LIN {X 0,Y 303.729,Z 621.055,A -85,B 0,C 180,E1 -15926.02,E2 -15926.02} C_VEL
LIN {X 0,Y 303.689,Z 622.489,A -85,B 0,C 180,E1 -15927.347,E2 -15927.347} C_VEL
LIN {X 0,Y 303.724,Z 623.5,A -85,B 0,C 180,E1 -15928.674,E2 -15928.674} C_VEL
LIN {X 0,Y 303.767,Z 624.114,A -85,B 0,C 180,E1 -15930,E2 -15930} C_VEL
LIN {X 0,Y 303.684,Z 624.33,A -85,B 0,C 180,E1 -15931.326,E2 -15931.326} C_VEL
LIN {X 0,Y 303.657,Z 624.123,A -85,B 0,C 180,E1 -15932.653,E2 -15932.653} C_VEL
LIN {X 0,Y 303.664,Z 623.508,A -85,B 0,C 180,E1 -15933.981,E2 -15933.981} C_VEL
LIN {X 0,Y 303.694,Z 622.179,A -85,B 0,C 180,E1 -15935.678,E2 -15935.678} C_VEL
LIN {X 0,Y 303.95,Z 619.276,A -85,B 0,C 180,E1 -15937.974,E2 -15937.974} C_VEL
LIN {X 0,Y 304.417,Z 615.707,A -85,B 0,C 180,E1 -15939.971,E2 -15939.971} C_VEL
LIN {X 0,Y 305.168,Z 611.059,A -85,B 0,C 180,E1 -15941.962,E2 -15941.962} C_VEL
LIN {X 0,Y 306.657,Z 604.076,A -85,B 0,C 180,E1 -15944.262,E2 -15944.262} C_VEL
LIN {X 0,Y 308.071,Z 596.828,A -85,B 0,C 180,E1 -15946.159,E2 -15946.159} C_VEL
LIN {X 0,Y 309.648,Z 588.913,A -85,B 0,C 180,E1 -15947.842,E2 -15947.842} C_VEL
LIN {X 0,Y 311.444,Z 579.671,A -85,B 0,C 180,E1 -15949.441,E2 -15949.441} C_VEL
LIN {X 0,Y 313.381,Z 569.416,A -85,B 0,C 180,E1 -15950.855,E2 -15950.855} C_VEL
LIN {X 0,Y 315.305,Z 558.079,A -85,B 0,C 180,E1 -15952.094,E2 -15952.094} C_VEL
LIN {X 0,Y 316.995,Z 546.32,A -85,B 0,C 180,E1 -15953.087,E2 -15953.087} C_VEL
LIN {X 0,Y 318.457,Z 533.399,A -85,B 0,C 180,E1 -15953.88,E2 -15953.88} C_VEL
LIN {X 0,Y 319.476,Z 519.67,A -85,B 0,C 180,E1 -15954.446,E2 -15954.446} C_VEL
LIN {X 0,Y 321.398,Z 456.74,A -85,B 0,C 180,E1 -15955.903,E2 -15955.903} C_VEL
LIN {X 0,Y 317.843,Z 434.507,A -85,B 0,C 180,E1 -15956.863,E2 -15956.863} C_VEL
LIN {X 0,Y 313.385,Z 414.246,A -85,B 0,C 180,E1 -15957.906,E2 -15957.906} C_VEL
LIN {X 0,Y 311.826,Z 410.324,A -85,B 0,C 180,E1 -15958.212,E2 -15958.212} C_VEL
LIN {X 0,Y 309.683,Z 400.252,A -85,B 0,C 180,E1 -15961.463,E2 -15961.463} C_VEL
LIN {X 0,Y 307.323,Z 390.367,A -85,B 0,C 180,E1 -15964.869,E2 -15964.869} C_VEL
LIN {X 0,Y 305.492,Z 383.429,A -85,B 0,C 180,E1 -15967.459,E2 -15967.459} C_VEL
LIN {X 0,Y 305.477,Z 383.421,A -85,B 0,C 180,E1 -15971.85,E2 -15971.85} C_VEL
LIN {X 0,Y 305.47,Z 383.432,A -85,B 0,C 180,E1 -15975.496,E2 -15975.496} C_VEL
LIN {X 0,Y 305.491,Z 383.43,A -85,B 0,C 180,E1 -15978.152,E2 -15978.152} C_VEL
LIN {X 0,Y 305.515,Z 383.43,A -85,B 0,C 180,E1 -15981.604,E2 -15981.604} C_VEL
LIN {X 0,Y 305.458,Z 383.435,A -85,B 0,C 180,E1 -15984.886,E2 -15984.886} C_VEL
LIN {X 0,Y 305.447,Z 383.436,A -85,B 0,C 180,E1 -15988.354,E2 -15988.354} C_VEL
LIN {X 0,Y 305.523,Z 383.423,A -85,B 0,C 180,E1 -15991.114,E2 -15991.114} C_VEL
LIN {X 0,Y 305.565,Z 383.413,A -85,B 0,C 180,E1 -15994.088,E2 -15994.088} C_VEL
LIN {X 0,Y 305.494,Z 383.421,A -85,B 0,C 180,E1 -15998.403,E2 -15998.403} C_VEL
LIN {X 0,Y 305.584,Z 383.42,A -85,B 0,C 180,E1 -16001.217,E2 -16001.217} C_VEL
LIN {X 0,Y 305.642,Z 383.415,A -85,B 0,C 180,E1 -16005.349,E2 -16005.349} C_VEL
LIN {X 0,Y 305.631,Z 383.413,A -85,B 0,C 180,E1 -16009.4,E2 -16009.4} C_VEL
LIN {X 0,Y 305.801,Z 383.38,A -85,B 0,C 180,E1 -16012.074,E2 -16012.074} C_VEL
LIN {X 0,Y 305.682,Z 383.407,A -85,B 0,C 180,E1 -16014.724,E2 -16014.724} C_VEL
LIN {X 0,Y 305.952,Z 383.367,A -85,B 0,C 180,E1 -16018.684,E2 -16018.684} C_VEL
LIN {X 0,Y 305.952,Z 383.368,A -85,B 0,C 180,E1 -16021.317,E2 -16021.317} C_VEL
LIN {X 0,Y 305.683,Z 383.409,A -85,B 0,C 180,E1 -16025.277,E2 -16025.277} C_VEL
LIN {X 0,Y 305.791,Z 383.386,A -85,B 0,C 180,E1 -16027.927,E2 -16027.927} C_VEL
LIN {X 0,Y 305.596,Z 383.407,A -85,B 0,C 180,E1 -16031.946,E2 -16031.946} C_VEL
LIN {X 0,Y 305.632,Z 383.412,A -85,B 0,C 180,E1 -16035.035,E2 -16035.035} C_VEL
LIN {X 0,Y 305.598,Z 383.413,A -85,B 0,C 180,E1 -16039.46,E2 -16039.46} C_VEL
LIN {X 0,Y 305.486,Z 383.429,A -85,B 0,C 180,E1 -16043.042,E2 -16043.042} C_VEL
LIN {X 0,Y 305.542,Z 383.425,A -85,B 0,C 180,E1 -16046.228,E2 -16046.228} C_VEL
LIN {X 0,Y 305.484,Z 383.434,A -85,B 0,C 180,E1 -16049.048,E2 -16049.048} C_VEL
LIN {X 0,Y 305.438,Z 383.44,A -85,B 0,C 180,E1 -16051.953,E2 -16051.953} C_VEL
LIN {X 0,Y 305.459,Z 383.421,A -85,B 0,C 180,E1 -16055.114,E2 -16055.114} C_VEL
LIN {X 0,Y 305.482,Z 383.434,A -85,B 0,C 180,E1 -16058.538,E2 -16058.538} C_VEL
LIN {X 0,Y 305.507,Z 383.421,A -85,B 0,C 180,E1 -16062.598,E2 -16062.598} C_VEL
LIN {X 0,Y 305.495,Z 383.468,A -85,B 0,C 180,E1 -16063.738,E2 -16063.738} C_VEL
LIN {X 0,Y 306.346,Z 387.007,A -85,B 0,C 180,E1 -16065.177,E2 -16065.177} C_VEL
LIN {X 0,Y 316.83,Z 407.501,A -85,B 0,C 180,E1 -16066.998,E2 -16066.998} C_VEL
LIN {X 0,Y 322.483,Z 420.618,A -85,B 0,C 180,E1 -16067.967,E2 -16067.967} C_VEL
LIN {X 0,Y 320.157,Z 493.367,A -85,B 0,C 180,E1 -16069.642,E2 -16069.642} C_VEL
LIN {X 0,Y 319.28,Z 507.116,A -85,B 0,C 180,E1 -16070.23,E2 -16070.23} C_VEL
LIN {X 0,Y 318.207,Z 518.81,A -85,B 0,C 180,E1 -16070.968,E2 -16070.968} C_VEL
LIN {X 0,Y 316.748,Z 530.87,A -85,B 0,C 180,E1 -16071.997,E2 -16071.997} C_VEL
LIN {X 0,Y 314.911,Z 542.97,A -85,B 0,C 180,E1 -16073.347,E2 -16073.347} C_VEL
LIN {X 0,Y 313.064,Z 553.69,A -85,B 0,C 180,E1 -16074.883,E2 -16074.883} C_VEL
LIN {X 0,Y 311.209,Z 563.2,A -85,B 0,C 180,E1 -16076.6,E2 -16076.6} C_VEL
LIN {X 0,Y 309.412,Z 571.675,A -85,B 0,C 180,E1 -16078.506,E2 -16078.506} C_VEL
LIN {X 0,Y 308.16,Z 577.308,A -85,B 0,C 180,E1 -16080.072,E2 -16080.072} C_VEL
LIN {X 0,Y 306.851,Z 582.985,A -85,B 0,C 180,E1 -16081.997,E2 -16081.997} C_VEL
LIN {X 0,Y 305.746,Z 587.839,A -85,B 0,C 180,E1 -16084.104,E2 -16084.104} C_VEL
LIN {X 0,Y 304.871,Z 591.45,A -85,B 0,C 180,E1 -16086.209,E2 -16086.209} C_VEL
LIN {X 0,Y 304.274,Z 593.945,A -85,B 0,C 180,E1 -16088.312,E2 -16088.312} C_VEL
LIN {X 0,Y 303.957,Z 595.012,A -85,B 0,C 180,E1 -16089.707,E2 -16089.707} C_VEL
LIN {X 0,Y 303.694,Z 595.804,A -85,B 0,C 180,E1 -16091.59,E2 -16091.59} C_VEL
LIN {X 0,Y 303.552,Z 595.674,A -85,B 0,C 180,E1 -16093.87,E2 -16093.87} C_VEL
LIN {X 0,Y 303.605,Z 594.112,A -85,B 0,C 180,E1 -16096.47,E2 -16096.47} C_VEL
LIN {X 0,Y 303.779,Z 592.511,A -85,B 0,C 180,E1 -16097.982,E2 -16097.982} C_VEL
LIN {X 0,Y 304.075,Z 589.456,A -85,B 0,C 180,E1 -16100.018,E2 -16100.018} C_VEL
LIN {X 0,Y 304.544,Z 585.326,A -85,B 0,C 180,E1 -16102.041,E2 -16102.041} C_VEL
LIN {X 0,Y 305.211,Z 579.004,A -85,B 0,C 180,E1 -16104.384,E2 -16104.384} C_VEL
LIN {X 0,Y 306.053,Z 572.12,A -85,B 0,C 180,E1 -16106.379,E2 -16106.379} C_VEL
LIN {X 0,Y 306.943,Z 565.092,A -85,B 0,C 180,E1 -16108.032,E2 -16108.032} C_VEL
LIN {X 0,Y 308.013,Z 556.621,A -85,B 0,C 180,E1 -16109.673,E2 -16109.673} C_VEL
LIN {X 0,Y 309.315,Z 546.128,A -85,B 0,C 180,E1 -16111.302,E2 -16111.302} C_VEL
LIN {X 0,Y 310.373,Z 535.779,A -85,B 0,C 180,E1 -16112.596,E2 -16112.596} C_VEL
LIN {X 0,Y 311.472,Z 524.411,A -85,B 0,C 180,E1 -16113.719,E2 -16113.719} C_VEL
LIN {X 0,Y 312.325,Z 512.792,A -85,B 0,C 180,E1 -16114.598,E2 -16114.598} C_VEL
LIN {X 0,Y 313.065,Z 499.421,A -85,B 0,C 180,E1 -16115.313,E2 -16115.313} C_VEL
LIN {X 0,Y 313.5,Z 486.358,A -85,B 0,C 180,E1 -16115.749,E2 -16115.749} C_VEL
LIN {X 0,Y 315.14,Z 413.753,A -85,B 0,C 180,E1 -16117.393,E2 -16117.393} C_VEL
LIN {X 0,Y 313.597,Z 407.414,A -85,B 0,C 180,E1 -16117.645,E2 -16117.645} C_VEL
LIN {X 0,Y 306.906,Z 387.756,A -85,B 0,C 180,E1 -16118.572,E2 -16118.572} C_VEL
LIN {X 0,Y 306.127,Z 385.487,A -85,B 0,C 180,E1 -16118.703,E2 -16118.703} C_VEL
LIN {X 0,Y 305.696,Z 383.41,A -85,B 0,C 180,E1 -16119.428,E2 -16119.428} C_VEL
LIN {X 0,Y 305.594,Z 383.423,A -85,B 0,C 180,E1 -16123.295,E2 -16123.295} C_VEL
LIN {X 0,Y 305.598,Z 383.417,A -85,B 0,C 180,E1 -16126.019,E2 -16126.019} C_VEL
LIN {X 0,Y 305.58,Z 383.422,A -85,B 0,C 180,E1 -16129.444,E2 -16129.444} C_VEL
LIN {X 0,Y 305.494,Z 383.432,A -85,B 0,C 180,E1 -16133.041,E2 -16133.041} C_VEL
LIN {X 0,Y 305.55,Z 383.422,A -85,B 0,C 180,E1 -16136.226,E2 -16136.226} C_VEL
LIN {X 0,Y 305.498,Z 383.432,A -85,B 0,C 180,E1 -16139.049,E2 -16139.049} C_VEL
LIN {X 0,Y 305.446,Z 383.434,A -85,B 0,C 180,E1 -16141.951,E2 -16141.951} C_VEL
LIN {X 0,Y 305.463,Z 383.438,A -85,B 0,C 180,E1 -16145.112,E2 -16145.112} C_VEL
LIN {X 0,Y 305.449,Z 383.435,A -85,B 0,C 180,E1 -16148.528,E2 -16148.528} C_VEL
LIN {X 0,Y 305.458,Z 383.433,A -85,B 0,C 180,E1 -16152.586,E2 -16152.586} C_VEL
LIN {X 0,Y 305.441,Z 383.434,A -85,B 0,C 180,E1 -16156.347,E2 -16156.347} C_VEL
LIN {X 0,Y 305.429,Z 383.435,A -85,B 0,C 180,E1 -16158.821,E2 -16158.821} C_VEL
LIN {X 0,Y 304.778,Z 383.518,A -85,B 0,C 180,E1 -16159.922,E2 -16159.922} C_VEL
LIN {X 0,Y 301.929,Z 383.872,A -85,B 0,C 180,E1 -16161.715,E2 -16161.715} C_VEL
LIN {X 0,Y 299.506,Z 384.176,A -85,B 0,C 180,E1 -16163.169,E2 -16163.169} C_VEL
LIN {X 0,Y 298.472,Z 384.303,A -85,B 0,C 180,E1 -16164.296,E2 -16164.296} C_VEL
LIN {X 0,Y 298.391,Z 384.309,A -85,B 0,C 180,E1 -16164.677,E2 -16164.677} C_VEL
LIN {X 0,Y 298.388,Z 384.317,A -85,B 0,C 180,E1 -16168.79,E2 -16168.79} C_VEL
LIN {X 0,Y 298.453,Z 384.305,A -85,B 0,C 180,E1 -16171.903,E2 -16171.903} C_VEL
LIN {X 0,Y 298.478,Z 384.305,A -85,B 0,C 180,E1 -16174.923,E2 -16174.923} C_VEL
LIN {X 0,Y 298.445,Z 384.307,A -85,B 0,C 180,E1 -16179.314,E2 -16179.314} C_VEL
LIN {X 0,Y 298.532,Z 384.296,A -85,B 0,C 180,E1 -16182.179,E2 -16182.179} C_VEL
LIN {X 0,Y 298.588,Z 384.29,A -85,B 0,C 180,E1 -16184.994,E2 -16184.994} C_VEL
LIN {X 0,Y 298.585,Z 384.288,A -85,B 0,C 180,E1 -16189.146,E2 -16189.146} C_VEL
LIN {X 0,Y 298.734,Z 384.269,A -85,B 0,C 180,E1 -16191.885,E2 -16191.885} C_VEL
LIN {X 0,Y 298.652,Z 384.285,A -85,B 0,C 180,E1 -16194.598,E2 -16194.598} C_VEL
LIN {X 0,Y 298.917,Z 384.246,A -85,B 0,C 180,E1 -16198.652,E2 -16198.652} C_VEL
LIN {X 0,Y 298.918,Z 384.236,A -85,B 0,C 180,E1 -16201.347,E2 -16201.347} C_VEL
LIN {X 0,Y 298.78,Z 384.267,A -85,B 0,C 180,E1 -16206.754,E2 -16206.754} C_VEL
LIN {X 0,Y 298.629,Z 384.283,A -85,B 0,C 180,E1 -16209.482,E2 -16209.482} C_VEL
LIN {X 0,Y 298.545,Z 384.294,A -85,B 0,C 180,E1 -16213.615,E2 -16213.615} C_VEL
LIN {X 0,Y 298.542,Z 384.298,A -85,B 0,C 180,E1 -16216.409,E2 -16216.409} C_VEL
LIN {X 0,Y 298.505,Z 384.299,A -85,B 0,C 180,E1 -16219.655,E2 -16219.655} C_VEL
LIN {X 0,Y 298.451,Z 384.305,A -85,B 0,C 180,E1 -16223.598,E2 -16223.598} C_VEL
LIN {X 0,Y 298.484,Z 384.304,A -85,B 0,C 180,E1 -16226.575,E2 -16226.575} C_VEL
LIN {X 0,Y 298.419,Z 384.311,A -85,B 0,C 180,E1 -16229.641,E2 -16229.641} C_VEL
LIN {X 0,Y 298.391,Z 384.315,A -85,B 0,C 180,E1 -16232.801,E2 -16232.801} C_VEL
LIN {X 0,Y 298.465,Z 384.306,A -85,B 0,C 180,E1 -16236.814,E2 -16236.814} C_VEL
LIN {X 0,Y 298.451,Z 384.308,A -85,B 0,C 180,E1 -16241.103,E2 -16241.103} C_VEL
LIN {X 0,Y 298.415,Z 384.312,A -85,B 0,C 180,E1 -16244.953,E2 -16244.953} C_VEL
LIN {X 0,Y 298.433,Z 384.309,A -85,B 0,C 180,E1 -16246.927,E2 -16246.927} C_VEL
LIN {X 0,Y 298.429,Z 384.31,A -85,B 0,C 180,E1 -16251,E2 -16251} C_VEL
LIN {X 0,Y 298.432,Z 384.314,A -85,B 0,C 180,E1 -16253.933,E2 -16253.933} C_VEL
LIN {X 0,Y 298.473,Z 384.367,A -85,B 0,C 180,E1 -16257.21,E2 -16257.21} C_VEL
LIN {X 0,Y 301.101,Z 396.996,A -85,B 0,C 180,E1 -16261.033,E2 -16261.033} C_VEL
LIN {X 0,Y 302.614,Z 405.329,A -85,B 0,C 180,E1 -16263.445,E2 -16263.445} C_VEL
LIN {X 0,Y 301.908,Z 411.128,A -85,B 0,C 180,E1 -16264.991,E2 -16264.991} C_VEL
LIN {X 0,Y 307.673,Z 456.514,A -85,B 0,C 180,E1 -16266.52,E2 -16266.52} C_VEL
LIN {X 0,Y 306.242,Z 519.842,A -85,B 0,C 180,E1 -16268.016,E2 -16268.016} C_VEL
LIN {X 0,Y 305.511,Z 533.114,A -85,B 0,C 180,E1 -16268.581,E2 -16268.581} C_VEL
LIN {X 0,Y 304.508,Z 545.884,A -85,B 0,C 180,E1 -16269.393,E2 -16269.393} C_VEL
LIN {X 0,Y 303.293,Z 557.205,A -85,B 0,C 180,E1 -16270.367,E2 -16270.367} C_VEL
LIN {X 0,Y 301.922,Z 568.932,A -85,B 0,C 180,E1 -16271.685,E2 -16271.685} C_VEL
LIN {X 0,Y 300.614,Z 579.485,A -85,B 0,C 180,E1 -16273.184,E2 -16273.184} C_VEL
LIN {X 0,Y 299.684,Z 588.254,A -85,B 0,C 180,E1 -16274.727,E2 -16274.727} C_VEL
LIN {X 0,Y 298.687,Z 596.06,A -85,B 0,C 180,E1 -16276.391,E2 -16276.391} C_VEL
LIN {X 0,Y 297.663,Z 603.777,A -85,B 0,C 180,E1 -16278.423,E2 -16278.423} C_VEL
LIN {X 0,Y 297.117,Z 609.987,A -85,B 0,C 180,E1 -16280.469,E2 -16280.469} C_VEL
LIN {X 0,Y 296.832,Z 614.9,A -85,B 0,C 180,E1 -16282.518,E2 -16282.518} C_VEL
LIN {X 0,Y 296.64,Z 618.653,A -85,B 0,C 180,E1 -16284.562,E2 -16284.562} C_VEL
LIN {X 0,Y 296.639,Z 620.586,A -85,B 0,C 180,E1 -16285.924,E2 -16285.924} C_VEL
LIN {X 0,Y 296.612,Z 622.071,A -85,B 0,C 180,E1 -16287.284,E2 -16287.284} C_VEL
LIN {X 0,Y 296.634,Z 623.105,A -85,B 0,C 180,E1 -16288.642,E2 -16288.642} C_VEL
LIN {X 0,Y 296.676,Z 623.743,A -85,B 0,C 180,E1 -16290,E2 -16290} C_VEL
LIN {X 0,Y 296.596,Z 623.983,A -85,B 0,C 180,E1 -16291.358,E2 -16291.358} C_VEL
LIN {X 0,Y 296.581,Z 623.823,A -85,B 0,C 180,E1 -16292.716,E2 -16292.716} C_VEL
LIN {X 0,Y 296.579,Z 623.233,A -85,B 0,C 180,E1 -16294.077,E2 -16294.077} C_VEL
LIN {X 0,Y 296.588,Z 622.122,A -85,B 0,C 180,E1 -16295.592,E2 -16295.592} C_VEL
LIN {X 0,Y 296.891,Z 619.103,A -85,B 0,C 180,E1 -16298.165,E2 -16298.165} C_VEL
LIN {X 0,Y 297.401,Z 615.582,A -85,B 0,C 180,E1 -16300.209,E2 -16300.209} C_VEL
LIN {X 0,Y 298.191,Z 610.993,A -85,B 0,C 180,E1 -16302.246,E2 -16302.246} C_VEL
LIN {X 0,Y 299.779,Z 604.087,A -85,B 0,C 180,E1 -16304.597,E2 -16304.597} C_VEL
LIN {X 0,Y 301.384,Z 596.293,A -85,B 0,C 180,E1 -16306.688,E2 -16306.688} C_VEL
LIN {X 0,Y 303.23,Z 587.415,A -85,B 0,C 180,E1 -16308.583,E2 -16308.583} C_VEL
LIN {X 0,Y 305.209,Z 577.869,A -85,B 0,C 180,E1 -16310.206,E2 -16310.206} C_VEL
LIN {X 0,Y 307.307,Z 567.319,A -85,B 0,C 180,E1 -16311.639,E2 -16311.639} C_VEL
LIN {X 0,Y 309.316,Z 555.556,A -85,B 0,C 180,E1 -16312.898,E2 -16312.898} C_VEL
LIN {X 0,Y 311.106,Z 542.995,A -85,B 0,C 180,E1 -16313.904,E2 -16313.904} C_VEL
LIN {X 0,Y 312.545,Z 529.756,A -85,B 0,C 180,E1 -16314.67,E2 -16314.67} C_VEL
LIN {X 0,Y 313.469,Z 516.138,A -85,B 0,C 180,E1 -16315.168,E2 -16315.168} C_VEL
LIN {X 0,Y 315.236,Z 457.401,A -85,B 0,C 180,E1 -16316.543,E2 -16316.543} C_VEL
LIN {X 0,Y 311.619,Z 435.007,A -85,B 0,C 180,E1 -16317.548,E2 -16317.548} C_VEL
LIN {X 0,Y 307.818,Z 417.418,A -85,B 0,C 180,E1 -16318.477,E2 -16318.477} C_VEL
LIN {X 0,Y 304.579,Z 409.918,A -85,B 0,C 180,E1 -16319.111,E2 -16319.111} C_VEL
LIN {X 0,Y 302.211,Z 399.013,A -85,B 0,C 180,E1 -16322.781,E2 -16322.781} C_VEL
LIN {X 0,Y 299.807,Z 389.463,A -85,B 0,C 180,E1 -16326.252,E2 -16326.252} C_VEL
LIN {X 0,Y 298.481,Z 384.296,A -85,B 0,C 180,E1 -16328.282,E2 -16328.282} C_VEL
LIN {X 0,Y 298.417,Z 384.304,A -85,B 0,C 180,E1 -16331.255,E2 -16331.255} C_VEL
LIN {X 0,Y 298.413,Z 384.312,A -85,B 0,C 180,E1 -16334.952,E2 -16334.952} C_VEL
LIN {X 0,Y 298.448,Z 384.309,A -85,B 0,C 180,E1 -16338.749,E2 -16338.749} C_VEL
LIN {X 0,Y 298.466,Z 384.301,A -85,B 0,C 180,E1 -16343.186,E2 -16343.186} C_VEL
LIN {X 0,Y 298.39,Z 384.31,A -85,B 0,C 180,E1 -16347.199,E2 -16347.199} C_VEL
LIN {X 0,Y 298.431,Z 384.304,A -85,B 0,C 180,E1 -16350.613,E2 -16350.613} C_VEL
LIN {X 0,Y 298.479,Z 384.297,A -85,B 0,C 180,E1 -16353.474,E2 -16353.474} C_VEL
LIN {X 0,Y 298.429,Z 384.309,A -85,B 0,C 180,E1 -16356.697,E2 -16356.697} C_VEL
LIN {X 0,Y 298.533,Z 384.298,A -85,B 0,C 180,E1 -16360.757,E2 -16360.757} C_VEL
LIN {X 0,Y 298.587,Z 384.291,A -85,B 0,C 180,E1 -16364.995,E2 -16364.995} C_VEL
LIN {X 0,Y 298.586,Z 384.288,A -85,B 0,C 180,E1 -16369.147,E2 -16369.147} C_VEL
LIN {X 0,Y 298.748,Z 384.26,A -85,B 0,C 180,E1 -16371.886,E2 -16371.886} C_VEL
LIN {X 0,Y 298.652,Z 384.282,A -85,B 0,C 180,E1 -16374.599,E2 -16374.599} C_VEL
LIN {X 0,Y 298.918,Z 384.243,A -85,B 0,C 180,E1 -16378.653,E2 -16378.653} C_VEL
LIN {X 0,Y 298.919,Z 384.244,A -85,B 0,C 180,E1 -16381.348,E2 -16381.348} C_VEL
LIN {X 0,Y 298.782,Z 384.259,A -85,B 0,C 180,E1 -16386.755,E2 -16386.755} C_VEL
LIN {X 0,Y 298.63,Z 384.288,A -85,B 0,C 180,E1 -16389.482,E2 -16389.482} C_VEL
LIN {X 0,Y 298.546,Z 384.298,A -85,B 0,C 180,E1 -16393.616,E2 -16393.616} C_VEL
LIN {X 0,Y 298.543,Z 384.287,A -85,B 0,C 180,E1 -16396.409,E2 -16396.409} C_VEL
LIN {X 0,Y 298.528,Z 384.292,A -85,B 0,C 180,E1 -16399.667,E2 -16399.667} C_VEL
LIN {X 0,Y 298.453,Z 384.301,A -85,B 0,C 180,E1 -16403.599,E2 -16403.599} C_VEL
LIN {X 0,Y 298.485,Z 384.302,A -85,B 0,C 180,E1 -16406.575,E2 -16406.575} C_VEL
LIN {X 0,Y 298.413,Z 384.311,A -85,B 0,C 180,E1 -16409.642,E2 -16409.642} C_VEL
LIN {X 0,Y 298.391,Z 384.31,A -85,B 0,C 180,E1 -16412.801,E2 -16412.801} C_VEL
LIN {X 0,Y 298.463,Z 384.311,A -85,B 0,C 180,E1 -16416.814,E2 -16416.814} C_VEL
LIN {X 0,Y 298.45,Z 384.305,A -85,B 0,C 180,E1 -16421.251,E2 -16421.251} C_VEL
LIN {X 0,Y 298.477,Z 384.421,A -85,B 0,C 180,E1 -16422.998,E2 -16422.998} C_VEL
LIN {X 0,Y 299.262,Z 387.536,A -85,B 0,C 180,E1 -16424.261,E2 -16424.261} C_VEL
LIN {X 0,Y 309.283,Z 406.733,A -85,B 0,C 180,E1 -16426.094,E2 -16426.094} C_VEL
LIN {X 0,Y 315.597,Z 420.647,A -85,B 0,C 180,E1 -16427.209,E2 -16427.209} C_VEL
LIN {X 0,Y 316.376,Z 422.565,A -85,B 0,C 180,E1 -16427.348,E2 -16427.348} C_VEL
LIN {X 0,Y 314.034,Z 493.114,A -85,B 0,C 180,E1 -16428.994,E2 -16428.994} C_VEL
LIN {X 0,Y 313.147,Z 506.803,A -85,B 0,C 180,E1 -16429.578,E2 -16429.578} C_VEL
LIN {X 0,Y 312.068,Z 518.11,A -85,B 0,C 180,E1 -16430.288,E2 -16430.288} C_VEL
LIN {X 0,Y 310.554,Z 530.224,A -85,B 0,C 180,E1 -16431.307,E2 -16431.307} C_VEL
LIN {X 0,Y 308.694,Z 542.145,A -85,B 0,C 180,E1 -16432.635,E2 -16432.635} C_VEL
LIN {X 0,Y 306.908,Z 552.293,A -85,B 0,C 180,E1 -16434.071,E2 -16434.071} C_VEL
LIN {X 0,Y 305.073,Z 561.288,A -85,B 0,C 180,E1 -16435.64,E2 -16435.64} C_VEL
LIN {X 0,Y 303.253,Z 569.426,A -85,B 0,C 180,E1 -16437.397,E2 -16437.397} C_VEL
LIN {X 0,Y 301.398,Z 577.606,A -85,B 0,C 180,E1 -16439.63,E2 -16439.63} C_VEL
LIN {X 0,Y 300.162,Z 582.555,A -85,B 0,C 180,E1 -16441.316,E2 -16441.316} C_VEL
LIN {X 0,Y 298.945,Z 587.577,A -85,B 0,C 180,E1 -16443.47,E2 -16443.47} C_VEL
LIN {X 0,Y 297.991,Z 591.349,A -85,B 0,C 180,E1 -16445.624,E2 -16445.624} C_VEL
LIN {X 0,Y 297.32,Z 593.99,A -85,B 0,C 180,E1 -16447.778,E2 -16447.778} C_VEL
LIN {X 0,Y 296.964,Z 595.187,A -85,B 0,C 180,E1 -16449.207,E2 -16449.207} C_VEL
LIN {X 0,Y 296.622,Z 596.138,A -85,B 0,C 180,E1 -16451.397,E2 -16451.397} C_VEL
LIN {X 0,Y 296.466,Z 596.099,A -85,B 0,C 180,E1 -16453.473,E2 -16453.473} C_VEL
LIN {X 0,Y 296.437,Z 595.539,A -85,B 0,C 180,E1 -16454.883,E2 -16454.883} C_VEL
LIN {X 0,Y 296.512,Z 594.496,A -85,B 0,C 180,E1 -16456.362,E2 -16456.362} C_VEL
LIN {X 0,Y 296.635,Z 593.172,A -85,B 0,C 180,E1 -16457.688,E2 -16457.688} C_VEL
LIN {X 0,Y 296.936,Z 590.247,A -85,B 0,C 180,E1 -16459.775,E2 -16459.775} C_VEL
LIN {X 0,Y 297.403,Z 586.269,A -85,B 0,C 180,E1 -16461.849,E2 -16461.849} C_VEL
LIN {X 0,Y 298.06,Z 580.156,A -85,B 0,C 180,E1 -16464.249,E2 -16464.249} C_VEL
LIN {X 0,Y 298.908,Z 573.449,A -85,B 0,C 180,E1 -16466.293,E2 -16466.293} C_VEL
LIN {X 0,Y 299.994,Z 565.128,A -85,B 0,C 180,E1 -16468.322,E2 -16468.322} C_VEL
LIN {X 0,Y 301.114,Z 556.577,A -85,B 0,C 180,E1 -16470,E2 -16470} C_VEL
LIN {X 0,Y 302.426,Z 546.35,A -85,B 0,C 180,E1 -16471.614,E2 -16471.614} C_VEL
LIN {X 0,Y 303.561,Z 535.545,A -85,B 0,C 180,E1 -16472.986,E2 -16472.986} C_VEL
LIN {X 0,Y 304.723,Z 524.005,A -85,B 0,C 180,E1 -16474.133,E2 -16474.133} C_VEL
LIN {X 0,Y 305.572,Z 512.108,A -85,B 0,C 180,E1 -16475.03,E2 -16475.03} C_VEL
LIN {X 0,Y 306.314,Z 499.225,A -85,B 0,C 180,E1 -16475.72,E2 -16475.72} C_VEL
LIN {X 0,Y 306.704,Z 487.342,A -85,B 0,C 180,E1 -16476.125,E2 -16476.125} C_VEL
LIN {X 0,Y 308.365,Z 414.381,A -85,B 0,C 180,E1 -16477.817,E2 -16477.817} C_VEL
LIN {X 0,Y 305.761,Z 405.34,A -85,B 0,C 180,E1 -16478.214,E2 -16478.214} C_VEL
LIN {X 0,Y 299.773,Z 388.209,A -85,B 0,C 180,E1 -16479.065,E2 -16479.065} C_VEL
LIN {X 0,Y 298.968,Z 385.779,A -85,B 0,C 180,E1 -16479.224,E2 -16479.224} C_VEL
LIN {X 0,Y 298.649,Z 384.288,A -85,B 0,C 180,E1 -16479.823,E2 -16479.823} C_VEL
LIN {X 0,Y 298.557,Z 384.298,A -85,B 0,C 180,E1 -16483.615,E2 -16483.615} C_VEL
LIN {X 0,Y 298.553,Z 384.295,A -85,B 0,C 180,E1 -16486.408,E2 -16486.408} C_VEL
LIN {X 0,Y 298.515,Z 384.301,A -85,B 0,C 180,E1 -16489.654,E2 -16489.654} C_VEL
LIN {X 0,Y 298.461,Z 384.303,A -85,B 0,C 180,E1 -16493.597,E2 -16493.597} C_VEL
LIN {X 0,Y 298.492,Z 384.302,A -85,B 0,C 180,E1 -16496.573,E2 -16496.573} C_VEL
LIN {X 0,Y 298.423,Z 384.312,A -85,B 0,C 180,E1 -16499.64,E2 -16499.64} C_VEL
LIN {X 0,Y 298.397,Z 384.314,A -85,B 0,C 180,E1 -16502.799,E2 -16502.799} C_VEL
LIN {X 0,Y 298.447,Z 384.308,A -85,B 0,C 180,E1 -16506.807,E2 -16506.807} C_VEL
LIN {X 0,Y 298.388,Z 384.316,A -85,B 0,C 180,E1 -16511.087,E2 -16511.087} C_VEL
LIN {X 0,Y 298.387,Z 384.318,A -85,B 0,C 180,E1 -16515.04,E2 -16515.04} C_VEL
LIN {X 0,Y 298.386,Z 384.317,A -85,B 0,C 180,E1 -16518.911,E2 -16518.911} C_VEL
LIN {X 0,Y 298.442,Z 384.309,A -85,B 0,C 180,E1 -16523.192,E2 -16523.192} C_VEL
LIN {X 0,Y 298.391,Z 384.309,A -85,B 0,C 180,E1 -16524.677,E2 -16524.677} C_VEL
LIN {X 0,Y 297.736,Z 384.396,A -85,B 0,C 180,E1 -16525.803,E2 -16525.803} C_VEL
LIN {X 0,Y 294.9,Z 384.748,A -85,B 0,C 180,E1 -16527.636,E2 -16527.636} C_VEL
LIN {X 0,Y 292.489,Z 385.049,A -85,B 0,C 180,E1 -16529.124,E2 -16529.124} C_VEL
LIN {X 0,Y 291.453,Z 385.176,A -85,B 0,C 180,E1 -16530.277,E2 -16530.277} C_VEL
LIN {X 0,Y 291.368,Z 385.187,A -85,B 0,C 180,E1 -16530.667,E2 -16530.667} C_VEL
LIN {X 0,Y 291.408,Z 385.184,A -85,B 0,C 180,E1 -16534.271,E2 -16534.271} C_VEL
LIN {X 0,Y 291.377,Z 385.187,A -85,B 0,C 180,E1 -16537.299,E2 -16537.299} C_VEL
LIN {X 0,Y 291.453,Z 385.179,A -85,B 0,C 180,E1 -16540.269,E2 -16540.269} C_VEL
LIN {X 0,Y 291.55,Z 385.166,A -85,B 0,C 180,E1 -16544.623,E2 -16544.623} C_VEL
LIN {X 0,Y 291.529,Z 385.169,A -85,B 0,C 180,E1 -16548.88,E2 -16548.88} C_VEL
LIN {X 0,Y 291.681,Z 385.147,A -85,B 0,C 180,E1 -16551.687,E2 -16551.687} C_VEL
LIN {X 0,Y 291.622,Z 385.16,A -85,B 0,C 180,E1 -16554.468,E2 -16554.468} C_VEL
LIN {X 0,Y 291.883,Z 385.121,A -85,B 0,C 180,E1 -16558.62,E2 -16558.62} C_VEL
LIN {X 0,Y 291.884,Z 385.11,A -85,B 0,C 180,E1 -16561.379,E2 -16561.379} C_VEL
LIN {X 0,Y 291.729,Z 385.144,A -85,B 0,C 180,E1 -16566.918,E2 -16566.918} C_VEL
LIN {X 0,Y 291.568,Z 385.163,A -85,B 0,C 180,E1 -16569.714,E2 -16569.714} C_VEL
LIN {X 0,Y 291.515,Z 385.171,A -85,B 0,C 180,E1 -16573.95,E2 -16573.95} C_VEL
LIN {X 0,Y 291.481,Z 385.174,A -85,B 0,C 180,E1 -16576.818,E2 -16576.818} C_VEL
LIN {X 0,Y 291.445,Z 385.18,A -85,B 0,C 180,E1 -16579.875,E2 -16579.875} C_VEL
LIN {X 0,Y 291.394,Z 385.188,A -85,B 0,C 180,E1 -16584.206,E2 -16584.206} C_VEL
LIN {X 0,Y 291.419,Z 385.182,A -85,B 0,C 180,E1 -16587.272,E2 -16587.272} C_VEL
LIN {X 0,Y 291.334,Z 385.196,A -85,B 0,C 180,E1 -16590.437,E2 -16590.437} C_VEL
LIN {X 0,Y 291.34,Z 385.195,A -85,B 0,C 180,E1 -16593.699,E2 -16593.699} C_VEL
LIN {X 0,Y 291.4,Z 385.186,A -85,B 0,C 180,E1 -16597.262,E2 -16597.262} C_VEL
LIN {X 0,Y 291.402,Z 385.187,A -85,B 0,C 180,E1 -16600.631,E2 -16600.631} C_VEL
LIN {X 0,Y 291.351,Z 385.194,A -85,B 0,C 180,E1 -16604.39,E2 -16604.39} C_VEL
LIN {X 0,Y 291.354,Z 385.192,A -85,B 0,C 180,E1 -16608.398,E2 -16608.398} C_VEL
LIN {X 0,Y 291.378,Z 385.189,A -85,B 0,C 180,E1 -16611.163,E2 -16611.163} C_VEL
LIN {X 0,Y 291.384,Z 385.19,A -85,B 0,C 180,E1 -16614.63,E2 -16614.63} C_VEL
LIN {X 0,Y 291.405,Z 385.278,A -85,B 0,C 180,E1 -16616.841,E2 -16616.841} C_VEL
LIN {X 0,Y 293.978,Z 397.522,A -85,B 0,C 180,E1 -16620.655,E2 -16620.655} C_VEL
LIN {X 0,Y 295.562,Z 405.864,A -85,B 0,C 180,E1 -16623.142,E2 -16623.142} C_VEL
LIN {X 0,Y 295.114,Z 410.849,A -85,B 0,C 180,E1 -16624.512,E2 -16624.512} C_VEL
LIN {X 0,Y 300.948,Z 457.099,A -85,B 0,C 180,E1 -16626.102,E2 -16626.102} C_VEL
LIN {X 0,Y 299.473,Z 520.035,A -85,B 0,C 180,E1 -16627.629,E2 -16627.629} C_VEL
LIN {X 0,Y 298.651,Z 533.894,A -85,B 0,C 180,E1 -16628.246,E2 -16628.246} C_VEL
LIN {X 0,Y 297.636,Z 546.347,A -85,B 0,C 180,E1 -16629.076,E2 -16629.076} C_VEL
LIN {X 0,Y 296.382,Z 557.455,A -85,B 0,C 180,E1 -16630.071,E2 -16630.071} C_VEL
LIN {X 0,Y 294.978,Z 569.076,A -85,B 0,C 180,E1 -16631.418,E2 -16631.418} C_VEL
LIN {X 0,Y 293.626,Z 579.546,A -85,B 0,C 180,E1 -16632.95,E2 -16632.95} C_VEL
LIN {X 0,Y 292.579,Z 588.958,A -85,B 0,C 180,E1 -16634.679,E2 -16634.679} C_VEL
LIN {X 0,Y 291.543,Z 596.673,A -85,B 0,C 180,E1 -16636.407,E2 -16636.407} C_VEL
LIN {X 0,Y 290.529,Z 604.217,A -85,B 0,C 180,E1 -16638.488,E2 -16638.488} C_VEL
LIN {X 0,Y 290.083,Z 609.363,A -85,B 0,C 180,E1 -16640.236,E2 -16640.236} C_VEL
LIN {X 0,Y 289.742,Z 614.336,A -85,B 0,C 180,E1 -16642.334,E2 -16642.334} C_VEL
LIN {X 0,Y 289.557,Z 618.149,A -85,B 0,C 180,E1 -16644.429,E2 -16644.429} C_VEL
LIN {X 0,Y 289.554,Z 620.11,A -85,B 0,C 180,E1 -16645.824,E2 -16645.824} C_VEL
LIN {X 0,Y 289.538,Z 621.639,A -85,B 0,C 180,E1 -16647.217,E2 -16647.217} C_VEL
LIN {X 0,Y 289.548,Z 622.707,A -85,B 0,C 180,E1 -16648.609,E2 -16648.609} C_VEL
LIN {X 0,Y 289.586,Z 623.37,A -85,B 0,C 180,E1 -16650,E2 -16650} C_VEL
LIN {X 0,Y 289.512,Z 623.635,A -85,B 0,C 180,E1 -16651.391,E2 -16651.391} C_VEL
LIN {X 0,Y 289.505,Z 623.513,A -85,B 0,C 180,E1 -16652.783,E2 -16652.783} C_VEL
LIN {X 0,Y 289.479,Z 622.959,A -85,B 0,C 180,E1 -16654.177,E2 -16654.177} C_VEL
LIN {X 0,Y 289.516,Z 622.006,A -85,B 0,C 180,E1 -16655.572,E2 -16655.572} C_VEL
LIN {X 0,Y 289.849,Z 618.918,A -85,B 0,C 180,E1 -16658.365,E2 -16658.365} C_VEL
LIN {X 0,Y 290.4,Z 615.443,A -85,B 0,C 180,E1 -16660.457,E2 -16660.457} C_VEL
LIN {X 0,Y 291.223,Z 610.912,A -85,B 0,C 180,E1 -16662.544,E2 -16662.544} C_VEL
LIN {X 0,Y 292.909,Z 604.103,A -85,B 0,C 180,E1 -16664.947,E2 -16664.947} C_VEL
LIN {X 0,Y 294.536,Z 596.624,A -85,B 0,C 180,E1 -16667.026,E2 -16667.026} C_VEL
LIN {X 0,Y 296.523,Z 587.65,A -85,B 0,C 180,E1 -16669.019,E2 -16669.019} C_VEL
LIN {X 0,Y 298.566,Z 578.246,A -85,B 0,C 180,E1 -16670.676,E2 -16670.676} C_VEL
LIN {X 0,Y 300.733,Z 567.843,A -85,B 0,C 180,E1 -16672.137,E2 -16672.137} C_VEL
LIN {X 0,Y 302.828,Z 556.319,A -85,B 0,C 180,E1 -16673.417,E2 -16673.417} C_VEL
LIN {X 0,Y 304.684,Z 544.156,A -85,B 0,C 180,E1 -16674.44,E2 -16674.44} C_VEL
LIN {X 0,Y 306.264,Z 530.685,A -85,B 0,C 180,E1 -16675.256,E2 -16675.256} C_VEL
LIN {X 0,Y 307.202,Z 518.211,A -85,B 0,C 180,E1 -16675.764,E2 -16675.764} C_VEL
LIN {X 0,Y 309.144,Z 458.455,A -85,B 0,C 180,E1 -16677.195,E2 -16677.195} C_VEL
LIN {X 0,Y 305.76,Z 437.076,A -85,B 0,C 180,E1 -16678.18,E2 -16678.18} C_VEL
LIN {X 0,Y 302.243,Z 420.535,A -85,B 0,C 180,E1 -16679.083,E2 -16679.083} C_VEL
LIN {X 0,Y 298.424,Z 412.243,A -85,B 0,C 180,E1 -16679.818,E2 -16679.818} C_VEL
LIN {X 0,Y 297.334,Z 409.414,A -85,B 0,C 180,E1 -16680.094,E2 -16680.094} C_VEL
LIN {X 0,Y 295.105,Z 399.586,A -85,B 0,C 180,E1 -16683.537,E2 -16683.537} C_VEL
LIN {X 0,Y 292.877,Z 390.777,A -85,B 0,C 180,E1 -16686.862,E2 -16686.862} C_VEL
LIN {X 0,Y 291.399,Z 385.18,A -85,B 0,C 180,E1 -16689.158,E2 -16689.158} C_VEL
LIN {X 0,Y 291.368,Z 385.189,A -85,B 0,C 180,E1 -16693.646,E2 -16693.646} C_VEL
LIN {X 0,Y 291.395,Z 385.185,A -85,B 0,C 180,E1 -16697.521,E2 -16697.521} C_VEL
LIN {X 0,Y 291.381,Z 385.188,A -85,B 0,C 180,E1 -16701.163,E2 -16701.163} C_VEL
LIN {X 0,Y 291.381,Z 385.189,A -85,B 0,C 180,E1 -16704.629,E2 -16704.629} C_VEL
LIN {X 0,Y 291.367,Z 385.192,A -85,B 0,C 180,E1 -16707.95,E2 -16707.95} C_VEL
LIN {X 0,Y 291.381,Z 385.184,A -85,B 0,C 180,E1 -16711.158,E2 -16711.158} C_VEL
LIN {X 0,Y 291.411,Z 385.176,A -85,B 0,C 180,E1 -16714.272,E2 -16714.272} C_VEL
LIN {X 0,Y 291.375,Z 385.184,A -85,B 0,C 180,E1 -16717.299,E2 -16717.299} C_VEL
LIN {X 0,Y 291.452,Z 385.181,A -85,B 0,C 180,E1 -16720.27,E2 -16720.27} C_VEL
LIN {X 0,Y 291.534,Z 385.169,A -85,B 0,C 180,E1 -16724.634,E2 -16724.634} C_VEL
LIN {X 0,Y 291.53,Z 385.165,A -85,B 0,C 180,E1 -16728.881,E2 -16728.881} C_VEL
LIN {X 0,Y 291.699,Z 385.139,A -85,B 0,C 180,E1 -16731.688,E2 -16731.688} C_VEL
LIN {X 0,Y 291.623,Z 385.158,A -85,B 0,C 180,E1 -16734.468,E2 -16734.468} C_VEL
LIN {X 0,Y 291.884,Z 385.119,A -85,B 0,C 180,E1 -16738.621,E2 -16738.621} C_VEL
LIN {X 0,Y 291.885,Z 385.119,A -85,B 0,C 180,E1 -16741.38,E2 -16741.38} C_VEL
LIN {X 0,Y 291.73,Z 385.136,A -85,B 0,C 180,E1 -16746.919,E2 -16746.919} C_VEL
LIN {X 0,Y 291.569,Z 385.166,A -85,B 0,C 180,E1 -16749.714,E2 -16749.714} C_VEL
LIN {X 0,Y 291.516,Z 385.172,A -85,B 0,C 180,E1 -16753.951,E2 -16753.951} C_VEL
LIN {X 0,Y 291.482,Z 385.168,A -85,B 0,C 180,E1 -16756.819,E2 -16756.819} C_VEL
LIN {X 0,Y 291.479,Z 385.169,A -85,B 0,C 180,E1 -16759.894,E2 -16759.894} C_VEL
LIN {X 0,Y 291.396,Z 385.179,A -85,B 0,C 180,E1 -16764.206,E2 -16764.206} C_VEL
LIN {X 0,Y 291.417,Z 385.18,A -85,B 0,C 180,E1 -16767.273,E2 -16767.273} C_VEL
LIN {X 0,Y 291.33,Z 385.192,A -85,B 0,C 180,E1 -16770.438,E2 -16770.438} C_VEL
LIN {X 0,Y 291.341,Z 385.178,A -85,B 0,C 180,E1 -16773.699,E2 -16773.699} C_VEL
LIN {X 0,Y 291.396,Z 385.187,A -85,B 0,C 180,E1 -16777.261,E2 -16777.261} C_VEL
LIN {X 0,Y 291.399,Z 385.189,A -85,B 0,C 180,E1 -16780.632,E2 -16780.632} C_VEL
LIN {X 0,Y 291.456,Z 385.37,A -85,B 0,C 180,E1 -16782.198,E2 -16782.198} C_VEL
LIN {X 0,Y 292.058,Z 387.811,A -85,B 0,C 180,E1 -16783.265,E2 -16783.265} C_VEL
LIN {X 0,Y 294.048,Z 391.492,A -85,B 0,C 180,E1 -16783.66,E2 -16783.66} C_VEL
LIN {X 0,Y 303.452,Z 409.285,A -85,B 0,C 180,E1 -16785.44,E2 -16785.44} C_VEL
LIN {X 0,Y 309.792,Z 423.207,A -85,B 0,C 180,E1 -16786.608,E2 -16786.608} C_VEL
LIN {X 0,Y 310.253,Z 424.406,A -85,B 0,C 180,E1 -16786.695,E2 -16786.695} C_VEL
LIN {X 0,Y 307.889,Z 493.966,A -85,B 0,C 180,E1 -16788.359,E2 -16788.359} C_VEL
LIN {X 0,Y 306.919,Z 507.621,A -85,B 0,C 180,E1 -16788.957,E2 -16788.957} C_VEL
LIN {X 0,Y 305.636,Z 520.407,A -85,B 0,C 180,E1 -16789.799,E2 -16789.799} C_VEL
LIN {X 0,Y 304.16,Z 531.281,A -85,B 0,C 180,E1 -16790.764,E2 -16790.764} C_VEL
LIN {X 0,Y 302.34,Z 542.476,A -85,B 0,C 180,E1 -16792.041,E2 -16792.041} C_VEL
LIN {X 0,Y 300.361,Z 553.111,A -85,B 0,C 180,E1 -16793.578,E2 -16793.578} C_VEL
LIN {X 0,Y 298.446,Z 562.003,A -85,B 0,C 180,E1 -16795.177,E2 -16795.177} C_VEL
LIN {X 0,Y 296.558,Z 570.067,A -85,B 0,C 180,E1 -16796.972,E2 -16796.972} C_VEL
LIN {X 0,Y 294.665,Z 577.909,A -85,B 0,C 180,E1 -16799.164,E2 -16799.164} C_VEL
LIN {X 0,Y 293.082,Z 584.03,A -85,B 0,C 180,E1 -16801.342,E2 -16801.342} C_VEL
LIN {X 0,Y 291.815,Z 588.841,A -85,B 0,C 180,E1 -16803.575,E2 -16803.575} C_VEL
LIN {X 0,Y 290.886,Z 592.312,A -85,B 0,C 180,E1 -16805.75,E2 -16805.75} C_VEL
LIN {X 0,Y 290.398,Z 594.028,A -85,B 0,C 180,E1 -16807.219,E2 -16807.219} C_VEL
LIN {X 0,Y 289.985,Z 595.309,A -85,B 0,C 180,E1 -16808.683,E2 -16808.683} C_VEL
LIN {X 0,Y 289.559,Z 596.47,A -85,B 0,C 180,E1 -16811.191,E2 -16811.191} C_VEL
LIN {X 0,Y 289.396,Z 596.476,A -85,B 0,C 180,E1 -16813.057,E2 -16813.057} C_VEL
LIN {X 0,Y 289.339,Z 596.035,A -85,B 0,C 180,E1 -16814.503,E2 -16814.503} C_VEL
LIN {X 0,Y 289.421,Z 594.882,A -85,B 0,C 180,E1 -16816.248,E2 -16816.248} C_VEL
LIN {X 0,Y 289.667,Z 592.082,A -85,B 0,C 180,E1 -16818.808,E2 -16818.808} C_VEL
LIN {X 0,Y 290.076,Z 588.604,A -85,B 0,C 180,E1 -16820.939,E2 -16820.939} C_VEL
LIN {X 0,Y 290.64,Z 584.027,A -85,B 0,C 180,E1 -16823.056,E2 -16823.056} C_VEL
LIN {X 0,Y 291.474,Z 577.09,A -85,B 0,C 180,E1 -16825.506,E2 -16825.506} C_VEL
LIN {X 0,Y 292.496,Z 569.564,A -85,B 0,C 180,E1 -16827.59,E2 -16827.59} C_VEL
LIN {X 0,Y 293.504,Z 561.893,A -85,B 0,C 180,E1 -16829.314,E2 -16829.314} C_VEL
LIN {X 0,Y 294.794,Z 552.546,A -85,B 0,C 180,E1 -16831.024,E2 -16831.024} C_VEL
LIN {X 0,Y 296.043,Z 542.343,A -85,B 0,C 180,E1 -16832.525,E2 -16832.525} C_VEL
LIN {X 0,Y 297.259,Z 530.633,A -85,B 0,C 180,E1 -16833.897,E2 -16833.897} C_VEL
LIN {X 0,Y 298.401,Z 518.486,A -85,B 0,C 180,E1 -16834.982,E2 -16834.982} C_VEL
LIN {X 0,Y 299.211,Z 505.803,A -85,B 0,C 180,E1 -16835.814,E2 -16835.814} C_VEL
LIN {X 0,Y 299.771,Z 492.647,A -85,B 0,C 180,E1 -16836.394,E2 -16836.394} C_VEL
LIN {X 0,Y 301.667,Z 415.122,A -85,B 0,C 180,E1 -16838.249,E2 -16838.249} C_VEL
LIN {X 0,Y 296.043,Z 397.771,A -85,B 0,C 180,E1 -16839.092,E2 -16839.092} C_VEL
LIN {X 0,Y 291.801,Z 386.118,A -85,B 0,C 180,E1 -16839.75,E2 -16839.75} C_VEL
LIN {X 0,Y 291.589,Z 385.166,A -85,B 0,C 180,E1 -16840.151,E2 -16840.151} C_VEL
LIN {X 0,Y 291.527,Z 385.172,A -85,B 0,C 180,E1 -16843.95,E2 -16843.95} C_VEL
LIN {X 0,Y 291.491,Z 385.176,A -85,B 0,C 180,E1 -16846.817,E2 -16846.817} C_VEL
LIN {X 0,Y 291.454,Z 385.179,A -85,B 0,C 180,E1 -16849.874,E2 -16849.874} C_VEL
LIN {X 0,Y 291.403,Z 385.179,A -85,B 0,C 180,E1 -16854.204,E2 -16854.204} C_VEL
LIN {X 0,Y 291.425,Z 385.186,A -85,B 0,C 180,E1 -16857.271,E2 -16857.271} C_VEL
LIN {X 0,Y 291.34,Z 385.193,A -85,B 0,C 180,E1 -16860.436,E2 -16860.436} C_VEL
LIN {X 0,Y 291.346,Z 385.193,A -85,B 0,C 180,E1 -16863.697,E2 -16863.697} C_VEL
LIN {X 0,Y 291.377,Z 385.191,A -85,B 0,C 180,E1 -16867.253,E2 -16867.253} C_VEL
LIN {X 0,Y 291.333,Z 385.194,A -85,B 0,C 180,E1 -16870.641,E2 -16870.641} C_VEL
LIN {X 0,Y 291.313,Z 385.195,A -85,B 0,C 180,E1 -16874.396,E2 -16874.396} C_VEL
LIN {X 0,Y 291.325,Z 385.193,A -85,B 0,C 180,E1 -16878.403,E2 -16878.403} C_VEL
LIN {X 0,Y 291.345,Z 385.193,A -85,B 0,C 180,E1 -16881.156,E2 -16881.156} C_VEL
LIN {X 0,Y 291.358,Z 385.191,A -85,B 0,C 180,E1 -16884.678,E2 -16884.678} C_VEL
LIN {X 0,Y 291.367,Z 385.188,A -85,B 0,C 180,E1 -16887.949,E2 -16887.949} C_VEL
LIN {X 0,Y 291.368,Z 385.187,A -85,B 0,C 180,E1 -16890.667,E2 -16890.667} C_VEL
LIN {X 0,Y 290.717,Z 385.273,A -85,B 0,C 180,E1 -16891.82,E2 -16891.82} C_VEL
LIN {X 0,Y 287.928,Z 385.627,A -85,B 0,C 180,E1 -16893.699,E2 -16893.699} C_VEL
LIN {X 0,Y 285.533,Z 385.924,A -85,B 0,C 180,E1 -16895.224,E2 -16895.224} C_VEL
LIN {X 0,Y 284.463,Z 386.051,A -85,B 0,C 180,E1 -16896.404,E2 -16896.404} C_VEL
LIN {X 0,Y 284.353,Z 386.062,A -85,B 0,C 180,E1 -16896.805,E2 -16896.805} C_VEL
LIN {X 0,Y 284.398,Z 386.056,A -85,B 0,C 180,E1 -16901.261,E2 -16901.261} C_VEL
LIN {X 0,Y 284.487,Z 386.044,A -85,B 0,C 180,E1 -16904.459,E2 -16904.459} C_VEL
LIN {X 0,Y 284.481,Z 386.049,A -85,B 0,C 180,E1 -16908.601,E2 -16908.601} C_VEL
LIN {X 0,Y 284.633,Z 386.024,A -85,B 0,C 180,E1 -16911.48,E2 -16911.48} C_VEL
LIN {X 0,Y 284.592,Z 386.034,A -85,B 0,C 180,E1 -16914.331,E2 -16914.331} C_VEL
LIN {X 0,Y 284.849,Z 385.996,A -85,B 0,C 180,E1 -16918.586,E2 -16918.586} C_VEL
LIN {X 0,Y 284.85,Z 385.985,A -85,B 0,C 180,E1 -16921.413,E2 -16921.413} C_VEL
LIN {X 0,Y 284.68,Z 386.022,A -85,B 0,C 180,E1 -16927.09,E2 -16927.09} C_VEL
LIN {X 0,Y 284.513,Z 386.043,A -85,B 0,C 180,E1 -16929.957,E2 -16929.957} C_VEL
LIN {X 0,Y 284.472,Z 386.051,A -85,B 0,C 180,E1 -16934.303,E2 -16934.303} C_VEL
LIN {X 0,Y 284.419,Z 386.052,A -85,B 0,C 180,E1 -16937.248,E2 -16937.248} C_VEL
LIN {X 0,Y 284.373,Z 386.063,A -85,B 0,C 180,E1 -16940.242,E2 -16940.242} C_VEL
LIN {X 0,Y 284.363,Z 386.061,A -85,B 0,C 180,E1 -16943.875,E2 -16943.875} C_VEL
LIN {X 0,Y 284.358,Z 386.065,A -85,B 0,C 180,E1 -16948.008,E2 -16948.008} C_VEL
LIN {X 0,Y 284.292,Z 386.071,A -85,B 0,C 180,E1 -16951.275,E2 -16951.275} C_VEL
LIN {X 0,Y 284.358,Z 386.063,A -85,B 0,C 180,E1 -16955.355,E2 -16955.355} C_VEL
LIN {X 0,Y 284.333,Z 386.071,A -85,B 0,C 180,E1 -16958.165,E2 -16958.165} C_VEL
LIN {X 0,Y 284.339,Z 386.07,A -85,B 0,C 180,E1 -16962.141,E2 -16962.141} C_VEL
LIN {X 0,Y 284.316,Z 386.072,A -85,B 0,C 180,E1 -16966.202,E2 -16966.202} C_VEL
LIN {X 0,Y 284.349,Z 386.064,A -85,B 0,C 180,E1 -16970.014,E2 -16970.014} C_VEL
LIN {X 0,Y 284.353,Z 386.065,A -85,B 0,C 180,E1 -16973.618,E2 -16973.618} C_VEL
LIN {X 0,Y 284.387,Z 386.09,A -85,B 0,C 180,E1 -16976.432,E2 -16976.432} C_VEL
LIN {X 0,Y 287.156,Z 399.444,A -85,B 0,C 180,E1 -16980.694,E2 -16980.694} C_VEL
LIN {X 0,Y 288.461,Z 406.389,A -85,B 0,C 180,E1 -16982.819,E2 -16982.819} C_VEL
LIN {X 0,Y 288.328,Z 410.442,A -85,B 0,C 180,E1 -16983.977,E2 -16983.977} C_VEL
LIN {X 0,Y 294.248,Z 457.16,A -85,B 0,C 180,E1 -16985.656,E2 -16985.656} C_VEL
LIN {X 0,Y 292.729,Z 519.468,A -85,B 0,C 180,E1 -16987.196,E2 -16987.196} C_VEL
LIN {X 0,Y 291.93,Z 533.118,A -85,B 0,C 180,E1 -16987.811,E2 -16987.811} C_VEL
LIN {X 0,Y 290.848,Z 545.706,A -85,B 0,C 180,E1 -16988.656,E2 -16988.656} C_VEL
LIN {X 0,Y 289.478,Z 557.696,A -85,B 0,C 180,E1 -16989.76,E2 -16989.76} C_VEL
LIN {X 0,Y 288.041,Z 569.218,A -85,B 0,C 180,E1 -16991.138,E2 -16991.138} C_VEL
LIN {X 0,Y 286.647,Z 579.597,A -85,B 0,C 180,E1 -16992.706,E2 -16992.706} C_VEL
LIN {X 0,Y 285.67,Z 588.098,A -85,B 0,C 180,E1 -16994.299,E2 -16994.299} C_VEL
LIN {X 0,Y 284.591,Z 595.903,A -85,B 0,C 180,E1 -16996.068,E2 -16996.068} C_VEL
LIN {X 0,Y 283.536,Z 603.525,A -85,B 0,C 180,E1 -16998.201,E2 -16998.201} C_VEL
LIN {X 0,Y 282.88,Z 610.574,A -85,B 0,C 180,E1 -17000.707,E2 -17000.707} C_VEL
LIN {X 0,Y 282.613,Z 615.213,A -85,B 0,C 180,E1 -17002.858,E2 -17002.858} C_VEL
LIN {X 0,Y 282.485,Z 617.761,A -85,B 0,C 180,E1 -17004.365,E2 -17004.365} C_VEL
LIN {X 0,Y 282.472,Z 619.634,A -85,B 0,C 180,E1 -17005.72,E2 -17005.72} C_VEL
LIN {X 0,Y 282.464,Z 621.195,A -85,B 0,C 180,E1 -17007.148,E2 -17007.148} C_VEL
LIN {X 0,Y 282.465,Z 622.31,A -85,B 0,C 180,E1 -17008.574,E2 -17008.574} C_VEL
LIN {X 0,Y 282.498,Z 622.997,A -85,B 0,C 180,E1 -17010,E2 -17010} C_VEL
LIN {X 0,Y 282.43,Z 623.287,A -85,B 0,C 180,E1 -17011.426,E2 -17011.426} C_VEL
LIN {X 0,Y 282.431,Z 623.192,A -85,B 0,C 180,E1 -17012.853,E2 -17012.853} C_VEL
LIN {X 0,Y 282.415,Z 621.94,A -85,B 0,C 180,E1 -17015.488,E2 -17015.488} C_VEL
LIN {X 0,Y 282.509,Z 620.438,A -85,B 0,C 180,E1 -17017.145,E2 -17017.145} C_VEL
LIN {X 0,Y 282.957,Z 617.685,A -85,B 0,C 180,E1 -17019.291,E2 -17019.291} C_VEL
LIN {X 0,Y 283.65,Z 613.934,A -85,B 0,C 180,E1 -17021.432,E2 -17021.432} C_VEL
LIN {X 0,Y 284.737,Z 609.093,A -85,B 0,C 180,E1 -17023.561,E2 -17023.561} C_VEL
LIN {X 0,Y 286.598,Z 601.899,A -85,B 0,C 180,E1 -17026.014,E2 -17026.014} C_VEL
LIN {X 0,Y 288.4,Z 593.992,A -85,B 0,C 180,E1 -17028.123,E2 -17028.123} C_VEL
LIN {X 0,Y 290.617,Z 584.367,A -85,B 0,C 180,E1 -17030.157,E2 -17030.157} C_VEL
LIN {X 0,Y 292.951,Z 574.341,A -85,B 0,C 180,E1 -17031.829,E2 -17031.829} C_VEL
LIN {X 0,Y 294.987,Z 564.444,A -85,B 0,C 180,E1 -17033.148,E2 -17033.148} C_VEL
LIN {X 0,Y 296.989,Z 553.717,A -85,B 0,C 180,E1 -17034.277,E2 -17034.277} C_VEL
LIN {X 0,Y 298.763,Z 541.956,A -85,B 0,C 180,E1 -17035.236,E2 -17035.236} C_VEL
LIN {X 0,Y 300.193,Z 529.366,A -85,B 0,C 180,E1 -17035.991,E2 -17035.991} C_VEL
LIN {X 0,Y 301.222,Z 516.051,A -85,B 0,C 180,E1 -17036.499,E2 -17036.499} C_VEL
LIN {X 0,Y 303.114,Z 459.405,A -85,B 0,C 180,E1 -17037.876,E2 -17037.876} C_VEL
LIN {X 0,Y 299.815,Z 438.434,A -85,B 0,C 180,E1 -17038.88,E2 -17038.88} C_VEL
LIN {X 0,Y 296.626,Z 423.392,A -85,B 0,C 180,E1 -17039.729,E2 -17039.729} C_VEL
LIN {X 0,Y 291.737,Z 412.869,A -85,B 0,C 180,E1 -17040.711,E2 -17040.711} C_VEL
LIN {X 0,Y 290.029,Z 409.059,A -85,B 0,C 180,E1 -17041.093,E2 -17041.093} C_VEL
LIN {X 0,Y 288.137,Z 400.752,A -85,B 0,C 180,E1 -17044.124,E2 -17044.124} C_VEL
LIN {X 0,Y 285.657,Z 390.71,A -85,B 0,C 180,E1 -17048.067,E2 -17048.067} C_VEL
LIN {X 0,Y 284.337,Z 386.07,A -85,B 0,C 180,E1 -17050.104,E2 -17050.104} C_VEL
LIN {X 0,Y 284.306,Z 386.073,A -85,B 0,C 180,E1 -17054.203,E2 -17054.203} C_VEL
LIN {X 0,Y 284.334,Z 386.065,A -85,B 0,C 180,E1 -17058.136,E2 -17058.136} C_VEL
LIN {X 0,Y 284.341,Z 386.064,A -85,B 0,C 180,E1 -17062.271,E2 -17062.271} C_VEL
LIN {X 0,Y 284.319,Z 386.068,A -85,B 0,C 180,E1 -17065.352,E2 -17065.352} C_VEL
LIN {X 0,Y 284.291,Z 386.07,A -85,B 0,C 180,E1 -17068.725,E2 -17068.725} C_VEL
LIN {X 0,Y 284.393,Z 386.057,A -85,B 0,C 180,E1 -17072.826,E2 -17072.826} C_VEL
LIN {X 0,Y 284.36,Z 386.062,A -85,B 0,C 180,E1 -17076.707,E2 -17076.707} C_VEL
LIN {X 0,Y 284.398,Z 386.058,A -85,B 0,C 180,E1 -17081.261,E2 -17081.261} C_VEL
LIN {X 0,Y 284.472,Z 386.048,A -85,B 0,C 180,E1 -17084.469,E2 -17084.469} C_VEL
LIN {X 0,Y 284.481,Z 386.042,A -85,B 0,C 180,E1 -17088.601,E2 -17088.601} C_VEL
LIN {X 0,Y 284.65,Z 386.019,A -85,B 0,C 180,E1 -17091.481,E2 -17091.481} C_VEL
LIN {X 0,Y 284.593,Z 386.033,A -85,B 0,C 180,E1 -17094.331,E2 -17094.331} C_VEL
LIN {X 0,Y 284.85,Z 385.996,A -85,B 0,C 180,E1 -17098.587,E2 -17098.587} C_VEL
LIN {X 0,Y 284.851,Z 385.995,A -85,B 0,C 180,E1 -17101.414,E2 -17101.414} C_VEL
LIN {X 0,Y 284.681,Z 386.013,A -85,B 0,C 180,E1 -17107.091,E2 -17107.091} C_VEL
LIN {X 0,Y 284.513,Z 386.044,A -85,B 0,C 180,E1 -17109.958,E2 -17109.958} C_VEL
LIN {X 0,Y 284.473,Z 386.05,A -85,B 0,C 180,E1 -17114.304,E2 -17114.304} C_VEL
LIN {X 0,Y 284.422,Z 386.05,A -85,B 0,C 180,E1 -17117.249,E2 -17117.249} C_VEL
LIN {X 0,Y 284.416,Z 386.048,A -85,B 0,C 180,E1 -17120.24,E2 -17120.24} C_VEL
LIN {X 0,Y 284.365,Z 386.055,A -85,B 0,C 180,E1 -17123.876,E2 -17123.876} C_VEL
LIN {X 0,Y 284.392,Z 386.054,A -85,B 0,C 180,E1 -17127.174,E2 -17127.174} C_VEL
LIN {X 0,Y 284.29,Z 386.073,A -85,B 0,C 180,E1 -17131.276,E2 -17131.276} C_VEL
LIN {X 0,Y 284.359,Z 386.05,A -85,B 0,C 180,E1 -17135.355,E2 -17135.355} C_VEL
LIN {X 0,Y 284.33,Z 386.066,A -85,B 0,C 180,E1 -17138.167,E2 -17138.167} C_VEL
LIN {X 0,Y 284.37,Z 386.155,A -85,B 0,C 180,E1 -17141.267,E2 -17141.267} C_VEL
LIN {X 0,Y 284.892,Z 388.156,A -85,B 0,C 180,E1 -17142.208,E2 -17142.208} C_VEL
LIN {X 0,Y 287.086,Z 392.07,A -85,B 0,C 180,E1 -17142.665,E2 -17142.665} C_VEL
LIN {X 0,Y 294.264,Z 405.314,A -85,B 0,C 180,E1 -17144.106,E2 -17144.106} C_VEL
LIN {X 0,Y 301.265,Z 419.509,A -85,B 0,C 180,E1 -17145.452,E2 -17145.452} C_VEL
LIN {X 0,Y 304.233,Z 426.33,A -85,B 0,C 180,E1 -17146.02,E2 -17146.02} C_VEL
LIN {X 0,Y 301.826,Z 493.875,A -85,B 0,C 180,E1 -17147.66,E2 -17147.66} C_VEL
LIN {X 0,Y 300.907,Z 507.262,A -85,B 0,C 180,E1 -17148.252,E2 -17148.252} C_VEL
LIN {X 0,Y 299.595,Z 519.596,A -85,B 0,C 180,E1 -17149.054,E2 -17149.054} C_VEL
LIN {X 0,Y 298.081,Z 530.652,A -85,B 0,C 180,E1 -17150.024,E2 -17150.024} C_VEL
LIN {X 0,Y 296.236,Z 541.757,A -85,B 0,C 180,E1 -17151.288,E2 -17151.288} C_VEL
LIN {X 0,Y 294.063,Z 552.797,A -85,B 0,C 180,E1 -17152.882,E2 -17152.882} C_VEL
LIN {X 0,Y 291.833,Z 562.706,A -85,B 0,C 180,E1 -17154.693,E2 -17154.693} C_VEL
LIN {X 0,Y 289.876,Z 570.708,A -85,B 0,C 180,E1 -17156.526,E2 -17156.526} C_VEL
LIN {X 0,Y 287.975,Z 578.191,A -85,B 0,C 180,E1 -17158.669,E2 -17158.669} C_VEL
LIN {X 0,Y 286.443,Z 583.622,A -85,B 0,C 180,E1 -17160.614,E2 -17160.614} C_VEL
LIN {X 0,Y 285.005,Z 588.907,A -85,B 0,C 180,E1 -17163.047,E2 -17163.047} C_VEL
LIN {X 0,Y 284.036,Z 592.248,A -85,B 0,C 180,E1 -17165.126,E2 -17165.126} C_VEL
LIN {X 0,Y 283.504,Z 594.074,A -85,B 0,C 180,E1 -17166.633,E2 -17166.633} C_VEL
LIN {X 0,Y 283.03,Z 595.422,A -85,B 0,C 180,E1 -17168.133,E2 -17168.133} C_VEL
LIN {X 0,Y 282.493,Z 596.803,A -85,B 0,C 180,E1 -17170.978,E2 -17170.978} C_VEL
LIN {X 0,Y 282.356,Z 596.851,A -85,B 0,C 180,E1 -17172.622,E2 -17172.622} C_VEL
LIN {X 0,Y 282.245,Z 596.478,A -85,B 0,C 180,E1 -17174.104,E2 -17174.104} C_VEL
LIN {X 0,Y 282.331,Z 595.266,A -85,B 0,C 180,E1 -17176.127,E2 -17176.127} C_VEL
LIN {X 0,Y 282.535,Z 592.784,A -85,B 0,C 180,E1 -17178.522,E2 -17178.522} C_VEL
LIN {X 0,Y 282.927,Z 589.446,A -85,B 0,C 180,E1 -17180.708,E2 -17180.708} C_VEL
LIN {X 0,Y 283.487,Z 585.016,A -85,B 0,C 180,E1 -17182.88,E2 -17182.88} C_VEL
LIN {X 0,Y 284.175,Z 579.388,A -85,B 0,C 180,E1 -17185.034,E2 -17185.034} C_VEL
LIN {X 0,Y 285.122,Z 572.354,A -85,B 0,C 180,E1 -17187.174,E2 -17187.174} C_VEL
LIN {X 0,Y 286.367,Z 563.523,A -85,B 0,C 180,E1 -17189.297,E2 -17189.297} C_VEL
LIN {X 0,Y 287.793,Z 553.484,A -85,B 0,C 180,E1 -17191.224,E2 -17191.224} C_VEL
LIN {X 0,Y 289.112,Z 543.226,A -85,B 0,C 180,E1 -17192.787,E2 -17192.787} C_VEL
LIN {X 0,Y 290.313,Z 531.884,A -85,B 0,C 180,E1 -17194.165,E2 -17194.165} C_VEL
LIN {X 0,Y 291.516,Z 520.054,A -85,B 0,C 180,E1 -17195.274,E2 -17195.274} C_VEL
LIN {X 0,Y 292.369,Z 507.125,A -85,B 0,C 180,E1 -17196.166,E2 -17196.166} C_VEL
LIN {X 0,Y 293.009,Z 493.306,A -85,B 0,C 180,E1 -17196.801,E2 -17196.801} C_VEL
LIN {X 0,Y 294.991,Z 416.315,A -85,B 0,C 180,E1 -17198.69,E2 -17198.69} C_VEL
LIN {X 0,Y 288.435,Z 396.576,A -85,B 0,C 180,E1 -17199.694,E2 -17199.694} C_VEL
LIN {X 0,Y 284.608,Z 386.483,A -85,B 0,C 180,E1 -17200.288,E2 -17200.288} C_VEL
LIN {X 0,Y 284.516,Z 386.048,A -85,B 0,C 180,E1 -17200.55,E2 -17200.55} C_VEL
LIN {X 0,Y 284.486,Z 386.049,A -85,B 0,C 180,E1 -17204.302,E2 -17204.302} C_VEL
LIN {X 0,Y 284.429,Z 386.058,A -85,B 0,C 180,E1 -17207.248,E2 -17207.248} C_VEL
LIN {X 0,Y 284.382,Z 386.059,A -85,B 0,C 180,E1 -17210.241,E2 -17210.241} C_VEL
LIN {X 0,Y 284.372,Z 386.055,A -85,B 0,C 180,E1 -17213.875,E2 -17213.875} C_VEL
LIN {X 0,Y 284.4,Z 386.062,A -85,B 0,C 180,E1 -17217.173,E2 -17217.173} C_VEL
LIN {X 0,Y 284.298,Z 386.073,A -85,B 0,C 180,E1 -17221.273,E2 -17221.273} C_VEL
LIN {X 0,Y 284.342,Z 386.066,A -85,B 0,C 180,E1 -17225.347,E2 -17225.347} C_VEL
LIN {X 0,Y 284.312,Z 386.067,A -85,B 0,C 180,E1 -17228.168,E2 -17228.168} C_VEL
LIN {X 0,Y 284.269,Z 386.07,A -85,B 0,C 180,E1 -17232.123,E2 -17232.123} C_VEL
LIN {X 0,Y 284.267,Z 386.071,A -85,B 0,C 180,E1 -17236.191,E2 -17236.191} C_VEL
LIN {X 0,Y 284.304,Z 386.068,A -85,B 0,C 180,E1 -17240.023,E2 -17240.023} C_VEL
LIN {X 0,Y 284.328,Z 386.064,A -85,B 0,C 180,E1 -17243.613,E2 -17243.613} C_VEL
LIN {X 0,Y 284.304,Z 386.07,A -85,B 0,C 180,E1 -17247.189,E2 -17247.189} C_VEL
LIN {X 0,Y 284.331,Z 386.062,A -85,B 0,C 180,E1 -17250.649,E2 -17250.649} C_VEL
LIN {X 0,Y 284.371,Z 386.06,A -85,B 0,C 180,E1 -17253.585,E2 -17253.585} C_VEL
LIN {X 0,Y 284.353,Z 386.062,A -85,B 0,C 180,E1 -17256.805,E2 -17256.805} C_VEL
LIN {X 0,Y 283.626,Z 386.152,A -85,B 0,C 180,E1 -17257.987,E2 -17257.987} C_VEL
LIN {X 0,Y 280.771,Z 386.508,A -85,B 0,C 180,E1 -17259.915,E2 -17259.915} C_VEL
LIN {X 0,Y 278.407,Z 386.802,A -85,B 0,C 180,E1 -17261.481,E2 -17261.481} C_VEL
LIN {X 0,Y 277.422,Z 386.926,A -85,B 0,C 180,E1 -17262.693,E2 -17262.693} C_VEL
LIN {X 0,Y 277.355,Z 386.928,A -85,B 0,C 180,E1 -17263.103,E2 -17263.103} C_VEL
LIN {X 0,Y 277.411,Z 386.93,A -85,B 0,C 180,E1 -17266.82,E2 -17266.82} C_VEL
LIN {X 0,Y 277.593,Z 386.902,A -85,B 0,C 180,E1 -17271.262,E2 -17271.262} C_VEL
LIN {X 0,Y 277.562,Z 386.909,A -85,B 0,C 180,E1 -17274.187,E2 -17274.187} C_VEL
LIN {X 0,Y 277.815,Z 386.872,A -85,B 0,C 180,E1 -17278.55,E2 -17278.55} C_VEL
LIN {X 0,Y 277.816,Z 386.859,A -85,B 0,C 180,E1 -17281.449,E2 -17281.449} C_VEL
LIN {X 0,Y 277.634,Z 386.899,A -85,B 0,C 180,E1 -17287.271,E2 -17287.271} C_VEL
LIN {X 0,Y 277.455,Z 386.924,A -85,B 0,C 180,E1 -17290.213,E2 -17290.213} C_VEL
LIN {X 0,Y 277.422,Z 386.928,A -85,B 0,C 180,E1 -17294.675,E2 -17294.675} C_VEL
LIN {X 0,Y 277.339,Z 386.935,A -85,B 0,C 180,E1 -17299.234,E2 -17299.234} C_VEL
LIN {X 0,Y 277.313,Z 386.941,A -85,B 0,C 180,E1 -17304.17,E2 -17304.17} C_VEL
LIN {X 0,Y 277.33,Z 386.937,A -85,B 0,C 180,E1 -17307.509,E2 -17307.509} C_VEL
LIN {X 0,Y 277.267,Z 386.948,A -85,B 0,C 180,E1 -17310.482,E2 -17310.482} C_VEL
LIN {X 0,Y 277.25,Z 386.951,A -85,B 0,C 180,E1 -17313.895,E2 -17313.895} C_VEL
LIN {X 0,Y 277.286,Z 386.946,A -85,B 0,C 180,E1 -17317.466,E2 -17317.466} C_VEL
LIN {X 0,Y 277.262,Z 386.949,A -85,B 0,C 180,E1 -17321.227,E2 -17321.227} C_VEL
LIN {X 0,Y 277.248,Z 386.95,A -85,B 0,C 180,E1 -17325.217,E2 -17325.217} C_VEL
LIN {X 0,Y 277.285,Z 386.944,A -85,B 0,C 180,E1 -17329.497,E2 -17329.497} C_VEL
LIN {X 0,Y 277.287,Z 386.943,A -85,B 0,C 180,E1 -17332.535,E2 -17332.535} C_VEL
LIN {X 0,Y 277.359,Z 387.109,A -85,B 0,C 180,E1 -17336.066,E2 -17336.066} C_VEL
LIN {X 0,Y 279.993,Z 399.804,A -85,B 0,C 180,E1 -17340.24,E2 -17340.24} C_VEL
LIN {X 0,Y 281.568,Z 408.288,A -85,B 0,C 180,E1 -17342.902,E2 -17342.902} C_VEL
LIN {X 0,Y 281.515,Z 410.218,A -85,B 0,C 180,E1 -17343.471,E2 -17343.471} C_VEL
LIN {X 0,Y 287.553,Z 457.785,A -85,B 0,C 180,E1 -17345.207,E2 -17345.207} C_VEL
LIN {X 0,Y 285.968,Z 519.412,A -85,B 0,C 180,E1 -17346.767,E2 -17346.767} C_VEL
LIN {X 0,Y 285.152,Z 533.003,A -85,B 0,C 180,E1 -17347.398,E2 -17347.398} C_VEL
LIN {X 0,Y 283.986,Z 546.039,A -85,B 0,C 180,E1 -17348.305,E2 -17348.305} C_VEL
LIN {X 0,Y 282.582,Z 557.877,A -85,B 0,C 180,E1 -17349.434,E2 -17349.434} C_VEL
LIN {X 0,Y 281.11,Z 569.306,A -85,B 0,C 180,E1 -17350.845,E2 -17350.845} C_VEL
LIN {X 0,Y 279.676,Z 579.593,A -85,B 0,C 180,E1 -17352.45,E2 -17352.45} C_VEL
LIN {X 0,Y 278.554,Z 588.866,A -85,B 0,C 180,E1 -17354.263,E2 -17354.263} C_VEL
LIN {X 0,Y 277.456,Z 596.487,A -85,B 0,C 180,E1 -17356.076,E2 -17356.076} C_VEL
LIN {X 0,Y 276.389,Z 603.949,A -85,B 0,C 180,E1 -17358.263,E2 -17358.263} C_VEL
LIN {X 0,Y 275.854,Z 609.943,A -85,B 0,C 180,E1 -17360.468,E2 -17360.468} C_VEL
LIN {X 0,Y 275.53,Z 614.65,A -85,B 0,C 180,E1 -17362.673,E2 -17362.673} C_VEL
LIN {X 0,Y 275.387,Z 617.577,A -85,B 0,C 180,E1 -17364.441,E2 -17364.441} C_VEL
LIN {X 0,Y 275.393,Z 620.744,A -85,B 0,C 180,E1 -17367.074,E2 -17367.074} C_VEL
LIN {X 0,Y 275.384,Z 621.908,A -85,B 0,C 180,E1 -17368.538,E2 -17368.538} C_VEL
LIN {X 0,Y 275.413,Z 622.624,A -85,B 0,C 180,E1 -17370,E2 -17370} C_VEL
LIN {X 0,Y 275.351,Z 622.94,A -85,B 0,C 180,E1 -17371.463,E2 -17371.463} C_VEL
LIN {X 0,Y 275.357,Z 622.87,A -85,B 0,C 180,E1 -17372.926,E2 -17372.926} C_VEL
LIN {X 0,Y 275.335,Z 621.809,A -85,B 0,C 180,E1 -17375.447,E2 -17375.447} C_VEL
LIN {X 0,Y 275.458,Z 620.223,A -85,B 0,C 180,E1 -17377.329,E2 -17377.329} C_VEL
LIN {X 0,Y 275.925,Z 617.526,A -85,B 0,C 180,E1 -17379.53,E2 -17379.53} C_VEL
LIN {X 0,Y 276.643,Z 613.835,A -85,B 0,C 180,E1 -17381.726,E2 -17381.726} C_VEL
LIN {X 0,Y 277.83,Z 609.059,A -85,B 0,C 180,E1 -17383.905,E2 -17383.905} C_VEL
LIN {X 0,Y 279.752,Z 601.935,A -85,B 0,C 180,E1 -17386.417,E2 -17386.417} C_VEL
LIN {X 0,Y 281.528,Z 594.666,A -85,B 0,C 180,E1 -17388.446,E2 -17388.446} C_VEL
LIN {X 0,Y 283.527,Z 586.404,A -85,B 0,C 180,E1 -17390.305,E2 -17390.305} C_VEL
LIN {X 0,Y 285.878,Z 576.876,A -85,B 0,C 180,E1 -17392.018,E2 -17392.018} C_VEL
LIN {X 0,Y 288.254,Z 566.341,A -85,B 0,C 180,E1 -17393.53,E2 -17393.53} C_VEL
LIN {X 0,Y 290.238,Z 556.215,A -85,B 0,C 180,E1 -17394.689,E2 -17394.689} C_VEL
LIN {X 0,Y 292.225,Z 544.311,A -85,B 0,C 180,E1 -17395.747,E2 -17395.747} C_VEL
LIN {X 0,Y 293.932,Z 531.142,A -85,B 0,C 180,E1 -17396.587,E2 -17396.587} C_VEL
LIN {X 0,Y 295.069,Z 517.537,A -85,B 0,C 180,E1 -17397.171,E2 -17397.171} C_VEL
LIN {X 0,Y 297.123,Z 460.237,A -85,B 0,C 180,E1 -17398.594,E2 -17398.594} C_VEL
LIN {X 0,Y 293.822,Z 439.436,A -85,B 0,C 180,E1 -17399.631,E2 -17399.631} C_VEL
LIN {X 0,Y 291.084,Z 426.311,A -85,B 0,C 180,E1 -17400.395,E2 -17400.395} C_VEL
LIN {X 0,Y 286.217,Z 416.033,A -85,B 0,C 180,E1 -17401.407,E2 -17401.407} C_VEL
LIN {X 0,Y 282.774,Z 408.623,A -85,B 0,C 180,E1 -17402.185,E2 -17402.185} C_VEL
LIN {X 0,Y 280.509,Z 399.092,A -85,B 0,C 180,E1 -17405.853,E2 -17405.853} C_VEL
LIN {X 0,Y 278.481,Z 391.249,A -85,B 0,C 180,E1 -17409.117,E2 -17409.117} C_VEL
LIN {X 0,Y 277.286,Z 386.936,A -85,B 0,C 180,E1 -17411.116,E2 -17411.116} C_VEL
LIN {X 0,Y 277.247,Z 386.947,A -85,B 0,C 180,E1 -17415.216,E2 -17415.216} C_VEL
LIN {X 0,Y 277.291,Z 386.943,A -85,B 0,C 180,E1 -17419.494,E2 -17419.494} C_VEL
LIN {X 0,Y 277.286,Z 386.941,A -85,B 0,C 180,E1 -17422.534,E2 -17422.534} C_VEL
LIN {X 0,Y 277.25,Z 386.942,A -85,B 0,C 180,E1 -17426.105,E2 -17426.105} C_VEL
LIN {X 0,Y 277.257,Z 386.941,A -85,B 0,C 180,E1 -17429.538,E2 -17429.538} C_VEL
LIN {X 0,Y 277.355,Z 386.932,A -85,B 0,C 180,E1 -17432.864,E2 -17432.864} C_VEL
LIN {X 0,Y 277.323,Z 386.94,A -85,B 0,C 180,E1 -17436.079,E2 -17436.079} C_VEL
LIN {X 0,Y 277.339,Z 386.938,A -85,B 0,C 180,E1 -17440.766,E2 -17440.766} C_VEL
LIN {X 0,Y 277.422,Z 386.93,A -85,B 0,C 180,E1 -17445.325,E2 -17445.325} C_VEL
LIN {X 0,Y 277.5,Z 386.92,A -85,B 0,C 180,E1 -17449.789,E2 -17449.789} C_VEL
LIN {X 0,Y 277.643,Z 386.886,A -85,B 0,C 180,E1 -17452.729,E2 -17452.729} C_VEL
LIN {X 0,Y 277.816,Z 386.871,A -85,B 0,C 180,E1 -17458.551,E2 -17458.551} C_VEL
LIN {X 0,Y 277.817,Z 386.871,A -85,B 0,C 180,E1 -17461.45,E2 -17461.45} C_VEL
LIN {X 0,Y 277.635,Z 386.89,A -85,B 0,C 180,E1 -17467.272,E2 -17467.272} C_VEL
LIN {X 0,Y 277.456,Z 386.923,A -85,B 0,C 180,E1 -17470.214,E2 -17470.214} C_VEL
LIN {X 0,Y 277.423,Z 386.929,A -85,B 0,C 180,E1 -17474.675,E2 -17474.675} C_VEL
LIN {X 0,Y 277.367,Z 386.931,A -85,B 0,C 180,E1 -17479.233,E2 -17479.233} C_VEL
LIN {X 0,Y 277.325,Z 386.931,A -85,B 0,C 180,E1 -17483.921,E2 -17483.921} C_VEL
LIN {X 0,Y 277.321,Z 386.935,A -85,B 0,C 180,E1 -17487.506,E2 -17487.506} C_VEL
LIN {X 0,Y 277.269,Z 386.943,A -85,B 0,C 180,E1 -17490.482,E2 -17490.482} C_VEL
LIN {X 0,Y 277.251,Z 386.931,A -85,B 0,C 180,E1 -17493.896,E2 -17493.896} C_VEL
LIN {X 0,Y 277.284,Z 386.944,A -85,B 0,C 180,E1 -17497.467,E2 -17497.467} C_VEL
LIN {X 0,Y 277.316,Z 387.047,A -85,B 0,C 180,E1 -17500.328,E2 -17500.328} C_VEL
LIN {X 0,Y 277.791,Z 388.734,A -85,B 0,C 180,E1 -17501.086,E2 -17501.086} C_VEL
LIN {X 0,Y 279.844,Z 392.347,A -85,B 0,C 180,E1 -17501.543,E2 -17501.543} C_VEL
LIN {X 0,Y 287.444,Z 405.855,A -85,B 0,C 180,E1 -17503.146,E2 -17503.146} C_VEL
LIN {X 0,Y 295.543,Z 422.082,A -85,B 0,C 180,E1 -17504.777,E2 -17504.777} C_VEL
LIN {X 0,Y 298.232,Z 428.279,A -85,B 0,C 180,E1 -17505.313,E2 -17505.313} C_VEL
LIN {X 0,Y 295.802,Z 494.355,A -85,B 0,C 180,E1 -17506.951,E2 -17506.951} C_VEL
LIN {X 0,Y 294.84,Z 507.704,A -85,B 0,C 180,E1 -17507.553,E2 -17507.553} C_VEL
LIN {X 0,Y 293.49,Z 519.862,A -85,B 0,C 180,E1 -17508.356,E2 -17508.356} C_VEL
LIN {X 0,Y 291.776,Z 531.795,A -85,B 0,C 180,E1 -17509.433,E2 -17509.433} C_VEL
LIN {X 0,Y 289.584,Z 543.944,A -85,B 0,C 180,E1 -17510.877,E2 -17510.877} C_VEL
LIN {X 0,Y 287.347,Z 554.735,A -85,B 0,C 180,E1 -17512.527,E2 -17512.527} C_VEL
LIN {X 0,Y 285.197,Z 563.69,A -85,B 0,C 180,E1 -17514.247,E2 -17514.247} C_VEL
LIN {X 0,Y 282.811,Z 572.774,A -85,B 0,C 180,E1 -17516.433,E2 -17516.433} C_VEL
LIN {X 0,Y 280.808,Z 580.151,A -85,B 0,C 180,E1 -17518.714,E2 -17518.714} C_VEL
LIN {X 0,Y 279.351,Z 585.087,A -85,B 0,C 180,E1 -17520.622,E2 -17520.622} C_VEL
LIN {X 0,Y 277.97,Z 589.737,A -85,B 0,C 180,E1 -17522.929,E2 -17522.929} C_VEL
LIN {X 0,Y 277.23,Z 592.154,A -85,B 0,C 180,E1 -17524.472,E2 -17524.472} C_VEL
LIN {X 0,Y 276.569,Z 594.279,A -85,B 0,C 180,E1 -17526.18,E2 -17526.18} C_VEL
LIN {X 0,Y 275.71,Z 596.527,A -85,B 0,C 180,E1 -17529.093,E2 -17529.093} C_VEL
LIN {X 0,Y 275.442,Z 597.135,A -85,B 0,C 180,E1 -17530.749,E2 -17530.749} C_VEL
LIN {X 0,Y 275.3,Z 597.227,A -85,B 0,C 180,E1 -17532.162,E2 -17532.162} C_VEL
LIN {X 0,Y 275.183,Z 596.917,A -85,B 0,C 180,E1 -17533.685,E2 -17533.685} C_VEL
LIN {X 0,Y 275.228,Z 595.638,A -85,B 0,C 180,E1 -17536.012,E2 -17536.012} C_VEL
LIN {X 0,Y 275.517,Z 592.55,A -85,B 0,C 180,E1 -17538.971,E2 -17538.971} C_VEL
LIN {X 0,Y 275.961,Z 588.996,A -85,B 0,C 180,E1 -17541.211,E2 -17541.211} C_VEL
LIN {X 0,Y 276.581,Z 584.325,A -85,B 0,C 180,E1 -17543.434,E2 -17543.434} C_VEL
LIN {X 0,Y 277.48,Z 577.278,A -85,B 0,C 180,E1 -17546.006,E2 -17546.006} C_VEL
LIN {X 0,Y 278.596,Z 569.647,A -85,B 0,C 180,E1 -17548.193,E2 -17548.193} C_VEL
LIN {X 0,Y 279.694,Z 561.848,A -85,B 0,C 180,E1 -17550,E2 -17550} C_VEL
LIN {X 0,Y 281.052,Z 552.598,A -85,B 0,C 180,E1 -17551.739,E2 -17551.739} C_VEL
LIN {X 0,Y 282.437,Z 541.704,A -85,B 0,C 180,E1 -17553.388,E2 -17553.388} C_VEL
LIN {X 0,Y 283.774,Z 529.881,A -85,B 0,C 180,E1 -17554.795,E2 -17554.795} C_VEL
LIN {X 0,Y 284.96,Z 517.212,A -85,B 0,C 180,E1 -17555.928,E2 -17555.928} C_VEL
LIN {X 0,Y 285.833,Z 504.583,A -85,B 0,C 180,E1 -17556.751,E2 -17556.751} C_VEL
LIN {X 0,Y 286.39,Z 491.899,A -85,B 0,C 180,E1 -17557.293,E2 -17557.293} C_VEL
LIN {X 0,Y 288.271,Z 417.508,A -85,B 0,C 180,E1 -17559.151,E2 -17559.151} C_VEL
LIN {X 0,Y 282.143,Z 399.104,A -85,B 0,C 180,E1 -17560.118,E2 -17560.118} C_VEL
LIN {X 0,Y 277.525,Z 387.362,A -85,B 0,C 180,E1 -17560.819,E2 -17560.819} C_VEL
LIN {X 0,Y 277.472,Z 386.926,A -85,B 0,C 180,E1 -17560.894,E2 -17560.894} C_VEL
LIN {X 0,Y 277.439,Z 386.928,A -85,B 0,C 180,E1 -17564.674,E2 -17564.674} C_VEL
LIN {X 0,Y 277.349,Z 386.94,A -85,B 0,C 180,E1 -17569.233,E2 -17569.233} C_VEL
LIN {X 0,Y 277.322,Z 386.932,A -85,B 0,C 180,E1 -17574.17,E2 -17574.17} C_VEL
LIN {X 0,Y 277.328,Z 386.94,A -85,B 0,C 180,E1 -17577.504,E2 -17577.504} C_VEL
LIN {X 0,Y 277.274,Z 386.946,A -85,B 0,C 180,E1 -17580.48,E2 -17580.48} C_VEL
LIN {X 0,Y 277.248,Z 386.948,A -85,B 0,C 180,E1 -17583.895,E2 -17583.895} C_VEL
LIN {X 0,Y 277.268,Z 386.946,A -85,B 0,C 180,E1 -17587.468,E2 -17587.468} C_VEL
LIN {X 0,Y 277.209,Z 386.952,A -85,B 0,C 180,E1 -17591.235,E2 -17591.235} C_VEL
LIN {X 0,Y 277.215,Z 386.952,A -85,B 0,C 180,E1 -17595.222,E2 -17595.222} C_VEL
LIN {X 0,Y 277.221,Z 386.951,A -85,B 0,C 180,E1 -17599.511,E2 -17599.511} C_VEL
LIN {X 0,Y 277.262,Z 386.945,A -85,B 0,C 180,E1 -17602.529,E2 -17602.529} C_VEL
LIN {X 0,Y 277.244,Z 386.948,A -85,B 0,C 180,E1 -17606.103,E2 -17606.103} C_VEL
LIN {X 0,Y 277.258,Z 386.943,A -85,B 0,C 180,E1 -17609.538,E2 -17609.538} C_VEL
LIN {X 0,Y 277.352,Z 386.939,A -85,B 0,C 180,E1 -17612.863,E2 -17612.863} C_VEL
LIN {X 0,Y 277.278,Z 386.938,A -85,B 0,C 180,E1 -17616.795,E2 -17616.795} C_VEL
LIN {X 0,Y 277.34,Z 386.939,A -85,B 0,C 180,E1 -17620.765,E2 -17620.765} C_VEL
LIN {X 0,Y 277.355,Z 386.928,A -85,B 0,C 180,E1 -17623.103,E2 -17623.103} C_VEL
LIN {X 0,Y 276.723,Z 387.011,A -85,B 0,C 180,E1 -17624.315,E2 -17624.315} C_VEL
LIN {X 0,Y 273.891,Z 387.366,A -85,B 0,C 180,E1 -17626.29,E2 -17626.29} C_VEL
LIN {X 0,Y 271.485,Z 387.667,A -85,B 0,C 180,E1 -17627.894,E2 -17627.894} C_VEL
LIN {X 0,Y 270.477,Z 387.79,A -85,B 0,C 180,E1 -17629.138,E2 -17629.138} C_VEL
LIN {X 0,Y 270.409,Z 387.796,A -85,B 0,C 180,E1 -17629.559,E2 -17629.559} C_VEL
LIN {X 0,Y 270.593,Z 387.777,A -85,B 0,C 180,E1 -17632.538,E2 -17632.538} C_VEL
LIN {X 0,Y 270.781,Z 387.747,A -85,B 0,C 180,E1 -17638.512,E2 -17638.512} C_VEL
LIN {X 0,Y 270.782,Z 387.734,A -85,B 0,C 180,E1 -17641.487,E2 -17641.487} C_VEL
LIN {X 0,Y 270.592,Z 387.776,A -85,B 0,C 180,E1 -17647.461,E2 -17647.461} C_VEL
LIN {X 0,Y 270.407,Z 387.8,A -85,B 0,C 180,E1 -17650.482,E2 -17650.482} C_VEL
LIN {X 0,Y 270.39,Z 387.802,A -85,B 0,C 180,E1 -17655.065,E2 -17655.065} C_VEL
LIN {X 0,Y 270.296,Z 387.813,A -85,B 0,C 180,E1 -17659.756,E2 -17659.756} C_VEL
LIN {X 0,Y 270.269,Z 387.819,A -85,B 0,C 180,E1 -17664.586,E2 -17664.586} C_VEL
LIN {X 0,Y 270.27,Z 387.819,A -85,B 0,C 180,E1 -17667.909,E2 -17667.909} C_VEL
LIN {X 0,Y 270.18,Z 387.829,A -85,B 0,C 180,E1 -17671.349,E2 -17671.349} C_VEL
LIN {X 0,Y 270.211,Z 387.826,A -85,B 0,C 180,E1 -17674.904,E2 -17674.904} C_VEL
LIN {X 0,Y 270.218,Z 387.827,A -85,B 0,C 180,E1 -17678.718,E2 -17678.718} C_VEL
LIN {X 0,Y 270.22,Z 387.827,A -85,B 0,C 180,E1 -17682.549,E2 -17682.549} C_VEL
LIN {X 0,Y 270.201,Z 387.827,A -85,B 0,C 180,E1 -17686.743,E2 -17686.743} C_VEL
LIN {X 0,Y 270.234,Z 387.822,A -85,B 0,C 180,E1 -17689.446,E2 -17689.446} C_VEL
LIN {X 0,Y 270.256,Z 387.822,A -85,B 0,C 180,E1 -17693.722,E2 -17693.722} C_VEL
LIN {X 0,Y 270.273,Z 387.829,A -85,B 0,C 180,E1 -17695.584,E2 -17695.584} C_VEL
LIN {X 0,Y 272.897,Z 400.439,A -85,B 0,C 180,E1 -17699.856,E2 -17699.856} C_VEL
LIN {X 0,Y 274.49,Z 408.785,A -85,B 0,C 180,E1 -17702.557,E2 -17702.557} C_VEL
LIN {X 0,Y 274.64,Z 410.192,A -85,B 0,C 180,E1 -17702.918,E2 -17702.918} C_VEL
LIN {X 0,Y 279.177,Z 444.862,A -85,B 0,C 180,E1 -17704.242,E2 -17704.242} C_VEL
LIN {X 0,Y 280.877,Z 459.826,A -85,B 0,C 180,E1 -17704.777,E2 -17704.777} C_VEL
LIN {X 0,Y 279.251,Z 518.995,A -85,B 0,C 180,E1 -17706.304,E2 -17706.304} C_VEL
LIN {X 0,Y 278.397,Z 532.89,A -85,B 0,C 180,E1 -17706.966,E2 -17706.966} C_VEL
LIN {X 0,Y 277.213,Z 545.334,A -85,B 0,C 180,E1 -17707.845,E2 -17707.845} C_VEL
LIN {X 0,Y 275.957,Z 556.473,A -85,B 0,C 180,E1 -17708.917,E2 -17708.917} C_VEL
LIN {X 0,Y 274.516,Z 566.775,A -85,B 0,C 180,E1 -17710.171,E2 -17710.171} C_VEL
LIN {X 0,Y 273.034,Z 577.479,A -85,B 0,C 180,E1 -17711.815,E2 -17711.815} C_VEL
LIN {X 0,Y 271.848,Z 586.227,A -85,B 0,C 180,E1 -17713.479,E2 -17713.479} C_VEL
LIN {X 0,Y 270.669,Z 594.264,A -85,B 0,C 180,E1 -17715.336,E2 -17715.336} C_VEL
LIN {X 0,Y 269.581,Z 602.103,A -85,B 0,C 180,E1 -17717.58,E2 -17717.58} C_VEL
LIN {X 0,Y 268.799,Z 609.297,A -85,B 0,C 180,E1 -17720.215,E2 -17720.215} C_VEL
LIN {X 0,Y 268.473,Z 614.073,A -85,B 0,C 180,E1 -17722.479,E2 -17722.479} C_VEL
LIN {X 0,Y 268.29,Z 617.384,A -85,B 0,C 180,E1 -17724.52,E2 -17724.52} C_VEL
LIN {X 0,Y 268.321,Z 620.287,A -85,B 0,C 180,E1 -17726.997,E2 -17726.997} C_VEL
LIN {X 0,Y 268.305,Z 621.49,A -85,B 0,C 180,E1 -17728.499,E2 -17728.499} C_VEL
LIN {X 0,Y 268.331,Z 622.249,A -85,B 0,C 180,E1 -17730,E2 -17730} C_VEL
LIN {X 0,Y 268.273,Z 622.592,A -85,B 0,C 180,E1 -17731.501,E2 -17731.501} C_VEL
LIN {X 0,Y 268.261,Z 622.547,A -85,B 0,C 180,E1 -17733.003,E2 -17733.003} C_VEL
LIN {X 0,Y 268.237,Z 621.669,A -85,B 0,C 180,E1 -17735.36,E2 -17735.36} C_VEL
LIN {X 0,Y 268.382,Z 620.008,A -85,B 0,C 180,E1 -17737.523,E2 -17737.523} C_VEL
LIN {X 0,Y 268.893,Z 617.368,A -85,B 0,C 180,E1 -17739.781,E2 -17739.781} C_VEL
LIN {X 0,Y 269.647,Z 613.736,A -85,B 0,C 180,E1 -17742.035,E2 -17742.035} C_VEL
LIN {X 0,Y 270.936,Z 609.027,A -85,B 0,C 180,E1 -17744.266,E2 -17744.266} C_VEL
LIN {X 0,Y 272.913,Z 601.983,A -85,B 0,C 180,E1 -17746.84,E2 -17746.84} C_VEL
LIN {X 0,Y 274.967,Z 594.187,A -85,B 0,C 180,E1 -17749.078,E2 -17749.078} C_VEL
LIN {X 0,Y 277.331,Z 584.923,A -85,B 0,C 180,E1 -17751.168,E2 -17751.168} C_VEL
LIN {X 0,Y 279.87,Z 575.165,A -85,B 0,C 180,E1 -17752.906,E2 -17752.906} C_VEL
LIN {X 0,Y 282.076,Z 565.633,A -85,B 0,C 180,E1 -17754.273,E2 -17754.273} C_VEL
LIN {X 0,Y 284.166,Z 555.423,A -85,B 0,C 180,E1 -17755.449,E2 -17755.449} C_VEL
LIN {X 0,Y 286.236,Z 543.33,A -85,B 0,C 180,E1 -17756.523,E2 -17756.523} C_VEL
LIN {X 0,Y 287.966,Z 529.95,A -85,B 0,C 180,E1 -17757.38,E2 -17757.38} C_VEL
LIN {X 0,Y 289.117,Z 516.901,A -85,B 0,C 180,E1 -17757.93,E2 -17757.93} C_VEL
LIN {X 0,Y 291.197,Z 461.364,A -85,B 0,C 180,E1 -17759.331,E2 -17759.331} C_VEL
LIN {X 0,Y 288.079,Z 441.313,A -85,B 0,C 180,E1 -17760.361,E2 -17760.361} C_VEL
LIN {X 0,Y 285.682,Z 429.475,A -85,B 0,C 180,E1 -17761.069,E2 -17761.069} C_VEL
LIN {X 0,Y 279.591,Z 416.586,A -85,B 0,C 180,E1 -17762.398,E2 -17762.398} C_VEL
LIN {X 0,Y 275.542,Z 408.201,A -85,B 0,C 180,E1 -17763.351,E2 -17763.351} C_VEL
LIN {X 0,Y 273.05,Z 398.043,A -85,B 0,C 180,E1 -17767.48,E2 -17767.48} C_VEL
LIN {X 0,Y 270.79,Z 389.757,A -85,B 0,C 180,E1 -17771.179,E2 -17771.179} C_VEL
LIN {X 0,Y 270.211,Z 387.812,A -85,B 0,C 180,E1 -17772.143,E2 -17772.143} C_VEL
LIN {X 0,Y 270.21,Z 387.827,A -85,B 0,C 180,E1 -17776.74,E2 -17776.74} C_VEL
LIN {X 0,Y 270.245,Z 387.821,A -85,B 0,C 180,E1 -17779.447,E2 -17779.447} C_VEL
LIN {X 0,Y 270.253,Z 387.816,A -85,B 0,C 180,E1 -17783.721,E2 -17783.721} C_VEL
LIN {X 0,Y 270.2,Z 387.82,A -85,B 0,C 180,E1 -17786.892,E2 -17786.892} C_VEL
LIN {X 0,Y 270.231,Z 387.815,A -85,B 0,C 180,E1 -17790.387,E2 -17790.387} C_VEL
LIN {X 0,Y 270.259,Z 387.81,A -85,B 0,C 180,E1 -17793.764,E2 -17793.764} C_VEL
LIN {X 0,Y 270.227,Z 387.82,A -85,B 0,C 180,E1 -17797.039,E2 -17797.039} C_VEL
LIN {X 0,Y 270.296,Z 387.816,A -85,B 0,C 180,E1 -17800.244,E2 -17800.244} C_VEL
LIN {X 0,Y 270.39,Z 387.803,A -85,B 0,C 180,E1 -17804.935,E2 -17804.935} C_VEL
LIN {X 0,Y 270.436,Z 387.797,A -85,B 0,C 180,E1 -17809.519,E2 -17809.519} C_VEL
LIN {X 0,Y 270.601,Z 387.763,A -85,B 0,C 180,E1 -17812.539,E2 -17812.539} C_VEL
LIN {X 0,Y 270.782,Z 387.746,A -85,B 0,C 180,E1 -17818.513,E2 -17818.513} C_VEL
LIN {X 0,Y 270.782,Z 387.746,A -85,B 0,C 180,E1 -17821.488,E2 -17821.488} C_VEL
LIN {X 0,Y 270.593,Z 387.767,A -85,B 0,C 180,E1 -17827.462,E2 -17827.462} C_VEL
LIN {X 0,Y 270.407,Z 387.801,A -85,B 0,C 180,E1 -17830.483,E2 -17830.483} C_VEL
LIN {X 0,Y 270.391,Z 387.8,A -85,B 0,C 180,E1 -17835.066,E2 -17835.066} C_VEL
LIN {X 0,Y 270.323,Z 387.805,A -85,B 0,C 180,E1 -17839.754,E2 -17839.754} C_VEL
LIN {X 0,Y 270.27,Z 387.812,A -85,B 0,C 180,E1 -17844.586,E2 -17844.586} C_VEL
LIN {X 0,Y 270.268,Z 387.815,A -85,B 0,C 180,E1 -17847.91,E2 -17847.91} C_VEL
LIN {X 0,Y 270.181,Z 387.831,A -85,B 0,C 180,E1 -17851.349,E2 -17851.349} C_VEL
LIN {X 0,Y 270.213,Z 387.808,A -85,B 0,C 180,E1 -17854.905,E2 -17854.905} C_VEL
LIN {X 0,Y 270.229,Z 387.825,A -85,B 0,C 180,E1 -17859.053,E2 -17859.053} C_VEL
LIN {X 0,Y 270.252,Z 387.963,A -85,B 0,C 180,E1 -17859.313,E2 -17859.313} C_VEL
LIN {X 0,Y 270.537,Z 389.048,A -85,B 0,C 180,E1 -17859.85,E2 -17859.85} C_VEL
LIN {X 0,Y 272.89,Z 393.051,A -85,B 0,C 180,E1 -17860.401,E2 -17860.401} C_VEL
LIN {X 0,Y 280.17,Z 405.554,A -85,B 0,C 180,E1 -17862.025,E2 -17862.025} C_VEL
LIN {X 0,Y 288.487,Z 421.865,A -85,B 0,C 180,E1 -17863.791,E2 -17863.791} C_VEL
LIN {X 0,Y 292.348,Z 430.494,A -85,B 0,C 180,E1 -17864.595,E2 -17864.595} C_VEL
LIN {X 0,Y 289.803,Z 495.065,A -85,B 0,C 180,E1 -17866.221,E2 -17866.221} C_VEL
LIN {X 0,Y 288.71,Z 508.734,A -85,B 0,C 180,E1 -17866.851,E2 -17866.851} C_VEL
LIN {X 0,Y 287.263,Z 521.289,A -85,B 0,C 180,E1 -17867.718,E2 -17867.718} C_VEL
LIN {X 0,Y 285.505,Z 532.924,A -85,B 0,C 180,E1 -17868.817,E2 -17868.817} C_VEL
LIN {X 0,Y 283.224,Z 544.928,A -85,B 0,C 180,E1 -17870.287,E2 -17870.287} C_VEL
LIN {X 0,Y 280.871,Z 555.552,A -85,B 0,C 180,E1 -17871.964,E2 -17871.964} C_VEL
LIN {X 0,Y 278.46,Z 565.096,A -85,B 0,C 180,E1 -17873.867,E2 -17873.867} C_VEL
LIN {X 0,Y 276.146,Z 573.443,A -85,B 0,C 180,E1 -17875.952,E2 -17875.952} C_VEL
LIN {X 0,Y 274.004,Z 580.893,A -85,B 0,C 180,E1 -17878.344,E2 -17878.344} C_VEL
LIN {X 0,Y 272.243,Z 586.456,A -85,B 0,C 180,E1 -17880.628,E2 -17880.628} C_VEL
LIN {X 0,Y 270.861,Z 590.861,A -85,B 0,C 180,E1 -17882.996,E2 -17882.996} C_VEL
LIN {X 0,Y 269.779,Z 594.08,A -85,B 0,C 180,E1 -17885.367,E2 -17885.367} C_VEL
LIN {X 0,Y 269.221,Z 595.644,A -85,B 0,C 180,E1 -17886.948,E2 -17886.948} C_VEL
LIN {X 0,Y 268.749,Z 596.709,A -85,B 0,C 180,E1 -17888.525,E2 -17888.525} C_VEL
LIN {X 0,Y 268.407,Z 597.464,A -85,B 0,C 180,E1 -17890.5,E2 -17890.5} C_VEL
LIN {X 0,Y 268.106,Z 597.357,A -85,B 0,C 180,E1 -17893.241,E2 -17893.241} C_VEL
LIN {X 0,Y 268.137,Z 596.015,A -85,B 0,C 180,E1 -17895.884,E2 -17895.884} C_VEL
LIN {X 0,Y 268.288,Z 594.176,A -85,B 0,C 180,E1 -17897.903,E2 -17897.903} C_VEL
LIN {X 0,Y 268.649,Z 591.107,A -85,B 0,C 180,E1 -17900.21,E2 -17900.21} C_VEL
LIN {X 0,Y 269.257,Z 586.557,A -85,B 0,C 180,E1 -17902.688,E2 -17902.688} C_VEL
LIN {X 0,Y 270.02,Z 580.626,A -85,B 0,C 180,E1 -17905.148,E2 -17905.148} C_VEL
LIN {X 0,Y 270.999,Z 573.733,A -85,B 0,C 180,E1 -17907.399,E2 -17907.399} C_VEL
LIN {X 0,Y 272.087,Z 566.684,A -85,B 0,C 180,E1 -17909.26,E2 -17909.26} C_VEL
LIN {X 0,Y 273.367,Z 558.191,A -85,B 0,C 180,E1 -17911.105,E2 -17911.105} C_VEL
LIN {X 0,Y 274.916,Z 547.666,A -85,B 0,C 180,E1 -17912.931,E2 -17912.931} C_VEL
LIN {X 0,Y 276.294,Z 535.877,A -85,B 0,C 180,E1 -17914.559,E2 -17914.559} C_VEL
LIN {X 0,Y 277.656,Z 523.94,A -85,B 0,C 180,E1 -17915.811,E2 -17915.811} C_VEL
LIN {X 0,Y 278.591,Z 511.641,A -85,B 0,C 180,E1 -17916.791,E2 -17916.791} C_VEL
LIN {X 0,Y 279.383,Z 499.094,A -85,B 0,C 180,E1 -17917.491,E2 -17917.491} C_VEL
LIN {X 0,Y 279.869,Z 484.81,A -85,B 0,C 180,E1 -17917.963,E2 -17917.963} C_VEL
LIN {X 0,Y 281.65,Z 419.066,A -85,B 0,C 180,E1 -17919.614,E2 -17919.614} C_VEL
LIN {X 0,Y 275.537,Z 400.695,A -85,B 0,C 180,E1 -17920.615,E2 -17920.615} C_VEL
LIN {X 0,Y 270.473,Z 388.124,A -85,B 0,C 180,E1 -17921.408,E2 -17921.408} C_VEL
LIN {X 0,Y 270.403,Z 387.808,A -85,B 0,C 180,E1 -17921.511,E2 -17921.511} C_VEL
LIN {X 0,Y 270.385,Z 387.806,A -85,B 0,C 180,E1 -17925.901,E2 -17925.901} C_VEL
LIN {X 0,Y 270.296,Z 387.815,A -85,B 0,C 180,E1 -17930.601,E2 -17930.601} C_VEL
LIN {X 0,Y 270.277,Z 387.81,A -85,B 0,C 180,E1 -17934.585,E2 -17934.585} C_VEL
LIN {X 0,Y 270.274,Z 387.817,A -85,B 0,C 180,E1 -17937.908,E2 -17937.908} C_VEL
LIN {X 0,Y 270.186,Z 387.83,A -85,B 0,C 180,E1 -17941.347,E2 -17941.347} C_VEL
LIN {X 0,Y 270.203,Z 387.829,A -85,B 0,C 180,E1 -17944.904,E2 -17944.904} C_VEL
LIN {X 0,Y 270.198,Z 387.827,A -85,B 0,C 180,E1 -17948.709,E2 -17948.709} C_VEL
LIN {X 0,Y 270.171,Z 387.831,A -85,B 0,C 180,E1 -17953.249,E2 -17953.249} C_VEL
LIN {X 0,Y 270.173,Z 387.828,A -85,B 0,C 180,E1 -17957.441,E2 -17957.441} C_VEL
LIN {X 0,Y 270.205,Z 387.824,A -85,B 0,C 180,E1 -17961.373,E2 -17961.373} C_VEL
LIN {X 0,Y 270.199,Z 387.829,A -85,B 0,C 180,E1 -17965.093,E2 -17965.093} C_VEL
LIN {X 0,Y 270.197,Z 387.824,A -85,B 0,C 180,E1 -17969.13,E2 -17969.13} C_VEL
LIN {X 0,Y 270.261,Z 387.818,A -85,B 0,C 180,E1 -17972.145,E2 -17972.145} C_VEL
LIN {X 0,Y 270.273,Z 387.813,A -85,B 0,C 180,E1 -17975.518,E2 -17975.518} C_VEL
LIN {X 0,Y 270.297,Z 387.814,A -85,B 0,C 180,E1 -17980.244,E2 -17980.244} C_VEL
LIN {X 0,Y 270.398,Z 387.802,A -85,B 0,C 180,E1 -17984.935,E2 -17984.935} C_VEL
LIN {X 0,Y 270.409,Z 387.796,A -85,B 0,C 180,E1 -17989.559,E2 -17989.559} C_VEL
LIN {X 0,Y 269.759,Z 387.879,A -85,B 0,C 180,E1 -17990.805,E2 -17990.805} C_VEL
LIN {X 0,Y 266.862,Z 388.243,A -85,B 0,C 180,E1 -17992.834,E2 -17992.834} C_VEL
LIN {X 0,Y 264.441,Z 388.546,A -85,B 0,C 180,E1 -17994.484,E2 -17994.484} C_VEL
LIN {X 0,Y 263.48,Z 388.661,A -85,B 0,C 180,E1 -17995.764,E2 -17995.764} C_VEL
LIN {X 0,Y 263.445,Z 388.662,A -85,B 0,C 180,E1 -17996.197,E2 -17996.197} C_VEL
LIN {X 0,Y 263.746,Z 388.623,A -85,B 0,C 180,E1 -17998.473,E2 -17998.473} C_VEL
LIN {X 0,Y 263.746,Z 388.608,A -85,B 0,C 180,E1 -18001.527,E2 -18001.527} C_VEL
LIN {X 0,Y 263.552,Z 388.653,A -85,B 0,C 180,E1 -18007.662,E2 -18007.662} C_VEL
LIN {X 0,Y 263.349,Z 388.677,A -85,B 0,C 180,E1 -18010.766,E2 -18010.766} C_VEL
LIN {X 0,Y 263.339,Z 388.68,A -85,B 0,C 180,E1 -18015.478,E2 -18015.478} C_VEL
LIN {X 0,Y 263.258,Z 388.694,A -85,B 0,C 180,E1 -18020.307,E2 -18020.307} C_VEL
LIN {X 0,Y 263.204,Z 388.697,A -85,B 0,C 180,E1 -18025.292,E2 -18025.292} C_VEL
LIN {X 0,Y 263.179,Z 388.702,A -85,B 0,C 180,E1 -18028.729,E2 -18028.729} C_VEL
LIN {X 0,Y 263.129,Z 388.71,A -85,B 0,C 180,E1 -18032.289,E2 -18032.289} C_VEL
LIN {X 0,Y 263.186,Z 388.704,A -85,B 0,C 180,E1 -18035.978,E2 -18035.978} C_VEL
LIN {X 0,Y 263.157,Z 388.709,A -85,B 0,C 180,E1 -18039.863,E2 -18039.863} C_VEL
LIN {X 0,Y 263.143,Z 388.711,A -85,B 0,C 180,E1 -18043.98,E2 -18043.98} C_VEL
LIN {X 0,Y 263.148,Z 388.706,A -85,B 0,C 180,E1 -18048.401,E2 -18048.401} C_VEL
LIN {X 0,Y 263.187,Z 388.702,A -85,B 0,C 180,E1 -18052.109,E2 -18052.109} C_VEL
LIN {X 0,Y 263.236,Z 388.797,A -85,B 0,C 180,E1 -18055.163,E2 -18055.163} C_VEL
LIN {X 0,Y 265.776,Z 400.914,A -85,B 0,C 180,E1 -18059.401,E2 -18059.401} C_VEL
LIN {X 0,Y 267.511,Z 409.8,A -85,B 0,C 180,E1 -18062.298,E2 -18062.298} C_VEL
LIN {X 0,Y 268.864,Z 416.042,A -85,B 0,C 180,E1 -18062.594,E2 -18062.594} C_VEL
LIN {X 0,Y 274.219,Z 459.873,A -85,B 0,C 180,E1 -18064.271,E2 -18064.271} C_VEL
LIN {X 0,Y 272.566,Z 517.75,A -85,B 0,C 180,E1 -18065.787,E2 -18065.787} C_VEL
LIN {X 0,Y 271.774,Z 531.208,A -85,B 0,C 180,E1 -18066.421,E2 -18066.421} C_VEL
LIN {X 0,Y 270.629,Z 543.473,A -85,B 0,C 180,E1 -18067.277,E2 -18067.277} C_VEL
LIN {X 0,Y 269.29,Z 555.024,A -85,B 0,C 180,E1 -18068.369,E2 -18068.369} C_VEL
LIN {X 0,Y 267.61,Z 566.857,A -85,B 0,C 180,E1 -18069.838,E2 -18069.838} C_VEL
LIN {X 0,Y 266.087,Z 577.495,A -85,B 0,C 180,E1 -18071.522,E2 -18071.522} C_VEL
LIN {X 0,Y 264.752,Z 587.072,A -85,B 0,C 180,E1 -18073.42,E2 -18073.42} C_VEL
LIN {X 0,Y 263.383,Z 596.265,A -85,B 0,C 180,E1 -18075.711,E2 -18075.711} C_VEL
LIN {X 0,Y 262.266,Z 603.649,A -85,B 0,C 180,E1 -18078.014,E2 -18078.014} C_VEL
LIN {X 0,Y 261.751,Z 608.652,A -85,B 0,C 180,E1 -18079.949,E2 -18079.949} C_VEL
LIN {X 0,Y 261.389,Z 613.494,A -85,B 0,C 180,E1 -18082.274,E2 -18082.274} C_VEL
LIN {X 0,Y 261.195,Z 617.187,A -85,B 0,C 180,E1 -18084.601,E2 -18084.601} C_VEL
LIN {X 0,Y 261.25,Z 619.831,A -85,B 0,C 180,E1 -18086.916,E2 -18086.916} C_VEL
LIN {X 0,Y 261.229,Z 621.062,A -85,B 0,C 180,E1 -18088.458,E2 -18088.458} C_VEL
LIN {X 0,Y 261.25,Z 621.873,A -85,B 0,C 180,E1 -18090,E2 -18090} C_VEL
LIN {X 0,Y 261.197,Z 622.244,A -85,B 0,C 180,E1 -18091.542,E2 -18091.542} C_VEL
LIN {X 0,Y 261.169,Z 622.225,A -85,B 0,C 180,E1 -18093.085,E2 -18093.085} C_VEL
LIN {X 0,Y 261.164,Z 621.498,A -85,B 0,C 180,E1 -18095.327,E2 -18095.327} C_VEL
LIN {X 0,Y 261.323,Z 619.795,A -85,B 0,C 180,E1 -18097.728,E2 -18097.728} C_VEL
LIN {X 0,Y 261.853,Z 617.215,A -85,B 0,C 180,E1 -18100.047,E2 -18100.047} C_VEL
LIN {X 0,Y 262.664,Z 613.65,A -85,B 0,C 180,E1 -18102.36,E2 -18102.36} C_VEL
LIN {X 0,Y 264.057,Z 609.012,A -85,B 0,C 180,E1 -18104.646,E2 -18104.646} C_VEL
LIN {X 0,Y 266.076,Z 602.043,A -85,B 0,C 180,E1 -18107.286,E2 -18107.286} C_VEL
LIN {X 0,Y 268.174,Z 594.62,A -85,B 0,C 180,E1 -18109.497,E2 -18109.497} C_VEL
LIN {X 0,Y 270.271,Z 586.924,A -85,B 0,C 180,E1 -18111.349,E2 -18111.349} C_VEL
LIN {X 0,Y 272.81,Z 577.713,A -85,B 0,C 180,E1 -18113.132,E2 -18113.132} C_VEL
LIN {X 0,Y 275.347,Z 567.496,A -85,B 0,C 180,E1 -18114.705,E2 -18114.705} C_VEL
LIN {X 0,Y 277.808,Z 556.204,A -85,B 0,C 180,E1 -18116.075,E2 -18116.075} C_VEL
LIN {X 0,Y 279.951,Z 544.512,A -85,B 0,C 180,E1 -18117.166,E2 -18117.166} C_VEL
LIN {X 0,Y 281.758,Z 531.754,A -85,B 0,C 180,E1 -18118.035,E2 -18118.035} C_VEL
LIN {X 0,Y 283.055,Z 518.131,A -85,B 0,C 180,E1 -18118.66,E2 -18118.66} C_VEL
LIN {X 0,Y 284.51,Z 484.123,A -85,B 0,C 180,E1 -18119.552,E2 -18119.552} C_VEL
LIN {X 0,Y 285.263,Z 461.951,A -85,B 0,C 180,E1 -18120.127,E2 -18120.127} C_VEL
LIN {X 0,Y 282.368,Z 443.026,A -85,B 0,C 180,E1 -18121.134,E2 -18121.134} C_VEL
LIN {X 0,Y 280.347,Z 432.72,A -85,B 0,C 180,E1 -18121.765,E2 -18121.765} C_VEL
LIN {X 0,Y 274.338,Z 419.973,A -85,B 0,C 180,E1 -18123.135,E2 -18123.135} C_VEL
LIN {X 0,Y 270.167,Z 411.808,A -85,B 0,C 180,E1 -18124.12,E2 -18124.12} C_VEL
LIN {X 0,Y 268.133,Z 407.633,A -85,B 0,C 180,E1 -18124.679,E2 -18124.679} C_VEL
LIN {X 0,Y 266.077,Z 398.98,A -85,B 0,C 180,E1 -18128.359,E2 -18128.359} C_VEL
LIN {X 0,Y 263.995,Z 391.601,A -85,B 0,C 180,E1 -18131.806,E2 -18131.806} C_VEL
LIN {X 0,Y 263.153,Z 388.697,A -85,B 0,C 180,E1 -18133.301,E2 -18133.301} C_VEL
LIN {X 0,Y 263.202,Z 388.696,A -85,B 0,C 180,E1 -18138.122,E2 -18138.122} C_VEL
LIN {X 0,Y 263.185,Z 388.7,A -85,B 0,C 180,E1 -18142.108,E2 -18142.108} C_VEL
LIN {X 0,Y 263.18,Z 388.695,A -85,B 0,C 180,E1 -18145.89,E2 -18145.89} C_VEL
LIN {X 0,Y 263.148,Z 388.698,A -85,B 0,C 180,E1 -18149.507,E2 -18149.507} C_VEL
LIN {X 0,Y 263.19,Z 388.695,A -85,B 0,C 180,E1 -18153.003,E2 -18153.003} C_VEL
LIN {X 0,Y 263.179,Z 388.701,A -85,B 0,C 180,E1 -18156.387,E2 -18156.387} C_VEL
LIN {X 0,Y 263.258,Z 388.689,A -85,B 0,C 180,E1 -18159.693,E2 -18159.693} C_VEL
LIN {X 0,Y 263.339,Z 388.681,A -85,B 0,C 180,E1 -18164.522,E2 -18164.522} C_VEL
LIN {X 0,Y 263.368,Z 388.675,A -85,B 0,C 180,E1 -18169.234,E2 -18169.234} C_VEL
LIN {X 0,Y 263.563,Z 388.639,A -85,B 0,C 180,E1 -18172.338,E2 -18172.338} C_VEL
LIN {X 0,Y 263.746,Z 388.622,A -85,B 0,C 180,E1 -18178.473,E2 -18178.473} C_VEL
LIN {X 0,Y 263.747,Z 388.622,A -85,B 0,C 180,E1 -18181.527,E2 -18181.527} C_VEL
LIN {X 0,Y 263.553,Z 388.644,A -85,B 0,C 180,E1 -18187.663,E2 -18187.663} C_VEL
LIN {X 0,Y 263.35,Z 388.676,A -85,B 0,C 180,E1 -18190.767,E2 -18190.767} C_VEL
LIN {X 0,Y 263.34,Z 388.675,A -85,B 0,C 180,E1 -18195.479,E2 -18195.479} C_VEL
LIN {X 0,Y 263.284,Z 388.68,A -85,B 0,C 180,E1 -18200.305,E2 -18200.305} C_VEL
LIN {X 0,Y 263.205,Z 388.698,A -85,B 0,C 180,E1 -18205.292,E2 -18205.292} C_VEL
LIN {X 0,Y 263.176,Z 388.704,A -85,B 0,C 180,E1 -18208.731,E2 -18208.731} C_VEL
LIN {X 0,Y 263.13,Z 388.707,A -85,B 0,C 180,E1 -18212.289,E2 -18212.289} C_VEL
LIN {X 0,Y 263.186,Z 388.694,A -85,B 0,C 180,E1 -18215.979,E2 -18215.979} C_VEL
LIN {X 0,Y 263.205,Z 388.81,A -85,B 0,C 180,E1 -18218.196,E2 -18218.196} C_VEL
LIN {X 0,Y 263.385,Z 389.681,A -85,B 0,C 180,E1 -18218.549,E2 -18218.549} C_VEL
LIN {X 0,Y 264.839,Z 392.448,A -85,B 0,C 180,E1 -18218.925,E2 -18218.925} C_VEL
LIN {X 0,Y 266.705,Z 395.029,A -85,B 0,C 180,E1 -18219.365,E2 -18219.365} C_VEL
LIN {X 0,Y 273.676,Z 406.728,A -85,B 0,C 180,E1 -18221,E2 -18221} C_VEL
LIN {X 0,Y 280.375,Z 419.427,A -85,B 0,C 180,E1 -18222.503,E2 -18222.503} C_VEL
LIN {X 0,Y 286.431,Z 432.454,A -85,B 0,C 180,E1 -18223.82,E2 -18223.82} C_VEL
LIN {X 0,Y 283.917,Z 494.968,A -85,B 0,C 180,E1 -18225.425,E2 -18225.425} C_VEL
LIN {X 0,Y 282.841,Z 508.512,A -85,B 0,C 180,E1 -18226.056,E2 -18226.056} C_VEL
LIN {X 0,Y 281.288,Z 521.264,A -85,B 0,C 180,E1 -18226.934,E2 -18226.934} C_VEL
LIN {X 0,Y 279.539,Z 532.378,A -85,B 0,C 180,E1 -18227.981,E2 -18227.981} C_VEL
LIN {X 0,Y 277.385,Z 543.521,A -85,B 0,C 180,E1 -18229.338,E2 -18229.338} C_VEL
LIN {X 0,Y 274.995,Z 554.254,A -85,B 0,C 180,E1 -18231,E2 -18231} C_VEL
LIN {X 0,Y 272.712,Z 562.977,A -85,B 0,C 180,E1 -18232.677,E2 -18232.677} C_VEL
LIN {X 0,Y 270.354,Z 571.268,A -85,B 0,C 180,E1 -18234.663,E2 -18234.663} C_VEL
LIN {X 0,Y 267.962,Z 579.183,A -85,B 0,C 180,E1 -18237.066,E2 -18237.066} C_VEL
LIN {X 0,Y 266.302,Z 584.328,A -85,B 0,C 180,E1 -18239.028,E2 -18239.028} C_VEL
LIN {X 0,Y 264.604,Z 589.324,A -85,B 0,C 180,E1 -18241.44,E2 -18241.44} C_VEL
LIN {X 0,Y 263.318,Z 593.078,A -85,B 0,C 180,E1 -18243.872,E2 -18243.872} C_VEL
LIN {X 0,Y 262.325,Z 595.705,A -85,B 0,C 180,E1 -18246.306,E2 -18246.306} C_VEL
LIN {X 0,Y 261.823,Z 596.892,A -85,B 0,C 180,E1 -18247.927,E2 -18247.927} C_VEL
LIN {X 0,Y 261.346,Z 597.8,A -85,B 0,C 180,E1 -18250.257,E2 -18250.257} C_VEL
LIN {X 0,Y 261.039,Z 597.782,A -85,B 0,C 180,E1 -18252.774,E2 -18252.774} C_VEL
LIN {X 0,Y 261.048,Z 596.391,A -85,B 0,C 180,E1 -18255.746,E2 -18255.746} C_VEL
LIN {X 0,Y 261.172,Z 594.826,A -85,B 0,C 180,E1 -18257.569,E2 -18257.569} C_VEL
LIN {X 0,Y 261.512,Z 591.885,A -85,B 0,C 180,E1 -18259.94,E2 -18259.94} C_VEL
LIN {X 0,Y 262.172,Z 587.108,A -85,B 0,C 180,E1 -18262.686,E2 -18262.686} C_VEL
LIN {X 0,Y 263.017,Z 580.728,A -85,B 0,C 180,E1 -18265.402,E2 -18265.402} C_VEL
LIN {X 0,Y 264.065,Z 573.778,A -85,B 0,C 180,E1 -18267.712,E2 -18267.712} C_VEL
LIN {X 0,Y 265.434,Z 565.06,A -85,B 0,C 180,E1 -18270,E2 -18270} C_VEL
LIN {X 0,Y 266.908,Z 555.569,A -85,B 0,C 180,E1 -18271.991,E2 -18271.991} C_VEL
LIN {X 0,Y 268.415,Z 545.076,A -85,B 0,C 180,E1 -18273.753,E2 -18273.753} C_VEL
LIN {X 0,Y 269.783,Z 533.905,A -85,B 0,C 180,E1 -18275.231,E2 -18275.231} C_VEL
LIN {X 0,Y 271.144,Z 521.366,A -85,B 0,C 180,E1 -18276.511,E2 -18276.511} C_VEL
LIN {X 0,Y 272.091,Z 508.608,A -85,B 0,C 180,E1 -18277.467,E2 -18277.467} C_VEL
LIN {X 0,Y 272.847,Z 494.986,A -85,B 0,C 180,E1 -18278.144,E2 -18278.144} C_VEL
LIN {X 0,Y 274.77,Z 432.247,A -85,B 0,C 180,E1 -18279.796,E2 -18279.796} C_VEL
LIN {X 0,Y 275.024,Z 420.544,A -85,B 0,C 180,E1 -18280.102,E2 -18280.102} C_VEL
LIN {X 0,Y 269.481,Z 403.811,A -85,B 0,C 180,E1 -18281.044,E2 -18281.044} C_VEL
LIN {X 0,Y 264.321,Z 391.435,A -85,B 0,C 180,E1 -18281.864,E2 -18281.864} C_VEL
LIN {X 0,Y 263.364,Z 388.683,A -85,B 0,C 180,E1 -18282.039,E2 -18282.039} C_VEL
LIN {X 0,Y 263.351,Z 388.682,A -85,B 0,C 180,E1 -18286.108,E2 -18286.108} C_VEL
LIN {X 0,Y 263.221,Z 388.697,A -85,B 0,C 180,E1 -18290.851,E2 -18290.851} C_VEL
LIN {X 0,Y 263.211,Z 388.695,A -85,B 0,C 180,E1 -18295.29,E2 -18295.29} C_VEL
LIN {X 0,Y 263.182,Z 388.701,A -85,B 0,C 180,E1 -18298.729,E2 -18298.729} C_VEL
LIN {X 0,Y 263.135,Z 388.705,A -85,B 0,C 180,E1 -18302.287,E2 -18302.287} C_VEL
LIN {X 0,Y 263.184,Z 388.7,A -85,B 0,C 180,E1 -18306.762,E2 -18306.762} C_VEL
LIN {X 0,Y 263.125,Z 388.705,A -85,B 0,C 180,E1 -18311.593,E2 -18311.593} C_VEL
LIN {X 0,Y 263.127,Z 388.704,A -85,B 0,C 180,E1 -18316.016,E2 -18316.016} C_VEL
LIN {X 0,Y 263.104,Z 388.709,A -85,B 0,C 180,E1 -18320.126,E2 -18320.126} C_VEL
LIN {X 0,Y 263.16,Z 388.7,A -85,B 0,C 180,E1 -18324.017,E2 -18324.017} C_VEL
LIN {X 0,Y 263.13,Z 388.705,A -85,B 0,C 180,E1 -18327.711,E2 -18327.711} C_VEL
LIN {X 0,Y 263.197,Z 388.697,A -85,B 0,C 180,E1 -18331.783,E2 -18331.783} C_VEL
LIN {X 0,Y 263.222,Z 388.693,A -85,B 0,C 180,E1 -18335.2,E2 -18335.2} C_VEL
LIN {X 0,Y 263.259,Z 388.689,A -85,B 0,C 180,E1 -18339.693,E2 -18339.693} C_VEL
LIN {X 0,Y 263.346,Z 388.677,A -85,B 0,C 180,E1 -18344.521,E2 -18344.521} C_VEL
LIN {X 0,Y 263.35,Z 388.676,A -85,B 0,C 180,E1 -18349.233,E2 -18349.233} C_VEL
LIN {X 0,Y 263.553,Z 388.652,A -85,B 0,C 180,E1 -18352.337,E2 -18352.337} C_VEL
LIN {X 0,Y 263.445,Z 388.662,A -85,B 0,C 180,E1 -18356.197,E2 -18356.197} C_VEL
LIN {X 0,Y 262.913,Z 388.729,A -85,B 0,C 180,E1 -18357.476,E2 -18357.476} C_VEL
LIN {X 0,Y 261.417,Z 388.912,A -85,B 0,C 180,E1 -18358.733,E2 -18358.733} C_VEL
LIN {X 0,Y 257.724,Z 389.359,A -85,B 0,C 180,E1 -18361.259,E2 -18361.259} C_VEL
LIN {X 0,Y 256.619,Z 389.5,A -85,B 0,C 180,E1 -18362.573,E2 -18362.573} C_VEL
LIN {X 0,Y 256.503,Z 389.519,A -85,B 0,C 180,E1 -18363.019,E2 -18363.019} C_VEL
LIN {X 0,Y 256.509,Z 389.531,A -85,B 0,C 180,E1 -18367.874,E2 -18367.874} C_VEL
LIN {X 0,Y 256.287,Z 389.56,A -85,B 0,C 180,E1 -18372.672,E2 -18372.672} C_VEL
LIN {X 0,Y 256.273,Z 389.563,A -85,B 0,C 180,E1 -18376.299,E2 -18376.299} C_VEL
LIN {X 0,Y 256.152,Z 389.576,A -85,B 0,C 180,E1 -18381.12,E2 -18381.12} C_VEL
LIN {X 0,Y 256.184,Z 389.572,A -85,B 0,C 180,E1 -18385.139,E2 -18385.139} C_VEL
LIN {X 0,Y 256.112,Z 389.582,A -85,B 0,C 180,E1 -18389.6,E2 -18389.6} C_VEL
LIN {X 0,Y 256.081,Z 389.586,A -85,B 0,C 180,E1 -18393.291,E2 -18393.291} C_VEL
LIN {X 0,Y 256.137,Z 389.581,A -85,B 0,C 180,E1 -18397.279,E2 -18397.279} C_VEL
LIN {X 0,Y 256.101,Z 389.586,A -85,B 0,C 180,E1 -18401.194,E2 -18401.194} C_VEL
LIN {X 0,Y 256.074,Z 389.589,A -85,B 0,C 180,E1 -18405.526,E2 -18405.526} C_VEL
LIN {X 0,Y 256.083,Z 389.584,A -85,B 0,C 180,E1 -18408.803,E2 -18408.803} C_VEL
LIN {X 0,Y 256.153,Z 389.575,A -85,B 0,C 180,E1 -18412.872,E2 -18412.872} C_VEL
LIN {X 0,Y 256.205,Z 389.711,A -85,B 0,C 180,E1 -18414.707,E2 -18414.707} C_VEL
LIN {X 0,Y 258.654,Z 401.379,A -85,B 0,C 180,E1 -18418.919,E2 -18418.919} C_VEL
LIN {X 0,Y 260.224,Z 409.145,A -85,B 0,C 180,E1 -18421.602,E2 -18421.602} C_VEL
LIN {X 0,Y 262.182,Z 415.988,A -85,B 0,C 180,E1 -18422.007,E2 -18422.007} C_VEL
LIN {X 0,Y 267.55,Z 460.103,A -85,B 0,C 180,E1 -18423.748,E2 -18423.748} C_VEL
LIN {X 0,Y 265.87,Z 517.565,A -85,B 0,C 180,E1 -18425.293,E2 -18425.293} C_VEL
LIN {X 0,Y 265.053,Z 530.969,A -85,B 0,C 180,E1 -18425.942,E2 -18425.942} C_VEL
LIN {X 0,Y 263.819,Z 543.78,A -85,B 0,C 180,E1 -18426.863,E2 -18426.863} C_VEL
LIN {X 0,Y 262.433,Z 555.157,A -85,B 0,C 180,E1 -18427.981,E2 -18427.981} C_VEL
LIN {X 0,Y 260.714,Z 566.892,A -85,B 0,C 180,E1 -18429.486,E2 -18429.486} C_VEL
LIN {X 0,Y 259.146,Z 577.468,A -85,B 0,C 180,E1 -18431.214,E2 -18431.214} C_VEL
LIN {X 0,Y 257.842,Z 586.105,A -85,B 0,C 180,E1 -18432.962,E2 -18432.962} C_VEL
LIN {X 0,Y 256.625,Z 594.053,A -85,B 0,C 180,E1 -18434.92,E2 -18434.92} C_VEL
LIN {X 0,Y 255.439,Z 601.783,A -85,B 0,C 180,E1 -18437.285,E2 -18437.285} C_VEL
LIN {X 0,Y 254.722,Z 607.996,A -85,B 0,C 180,E1 -18439.669,E2 -18439.669} C_VEL
LIN {X 0,Y 254.331,Z 612.909,A -85,B 0,C 180,E1 -18442.058,E2 -18442.058} C_VEL
LIN {X 0,Y 254.1,Z 616.986,A -85,B 0,C 180,E1 -18444.687,E2 -18444.687} C_VEL
LIN {X 0,Y 254.157,Z 619.369,A -85,B 0,C 180,E1 -18446.83,E2 -18446.83} C_VEL
LIN {X 0,Y 254.155,Z 620.63,A -85,B 0,C 180,E1 -18448.415,E2 -18448.415} C_VEL
LIN {X 0,Y 254.172,Z 621.485,A -85,B 0,C 180,E1 -18450,E2 -18450} C_VEL
LIN {X 0,Y 254.122,Z 621.895,A -85,B 0,C 180,E1 -18451.585,E2 -18451.585} C_VEL
LIN {X 0,Y 254.08,Z 621.903,A -85,B 0,C 180,E1 -18453.171,E2 -18453.171} C_VEL
LIN {X 0,Y 254.086,Z 621.337,A -85,B 0,C 180,E1 -18455.279,E2 -18455.279} C_VEL
LIN {X 0,Y 254.264,Z 619.587,A -85,B 0,C 180,E1 -18457.944,E2 -18457.944} C_VEL
LIN {X 0,Y 254.82,Z 617.063,A -85,B 0,C 180,E1 -18460.327,E2 -18460.327} C_VEL
LIN {X 0,Y 255.696,Z 613.551,A -85,B 0,C 180,E1 -18462.702,E2 -18462.702} C_VEL
LIN {X 0,Y 257.165,Z 608.981,A -85,B 0,C 180,E1 -18465.047,E2 -18465.047} C_VEL
LIN {X 0,Y 258.955,Z 603.22,A -85,B 0,C 180,E1 -18467.369,E2 -18467.369} C_VEL
LIN {X 0,Y 260.915,Z 596.689,A -85,B 0,C 180,E1 -18469.48,E2 -18469.48} C_VEL
LIN {X 0,Y 263.225,Z 588.793,A -85,B 0,C 180,E1 -18471.538,E2 -18471.538} C_VEL
LIN {X 0,Y 265.771,Z 580.042,A -85,B 0,C 180,E1 -18473.369,E2 -18473.369} C_VEL
LIN {X 0,Y 268.63,Z 569.307,A -85,B 0,C 180,E1 -18475.159,E2 -18475.159} C_VEL
LIN {X 0,Y 271.146,Z 558.605,A -85,B 0,C 180,E1 -18476.558,E2 -18476.558} C_VEL
LIN {X 0,Y 273.546,Z 546.633,A -85,B 0,C 180,E1 -18477.753,E2 -18477.753} C_VEL
LIN {X 0,Y 275.527,Z 534.201,A -85,B 0,C 180,E1 -18478.676,E2 -18478.676} C_VEL
LIN {X 0,Y 276.908,Z 521.733,A -85,B 0,C 180,E1 -18479.329,E2 -18479.329} C_VEL
LIN {X 0,Y 277.822,Z 506.606,A -85,B 0,C 180,E1 -18479.799,E2 -18479.799} C_VEL
LIN {X 0,Y 279.478,Z 463.019,A -85,B 0,C 180,E1 -18480.932,E2 -18480.932} C_VEL
LIN {X 0,Y 276.768,Z 445.085,A -85,B 0,C 180,E1 -18481.919,E2 -18481.919} C_VEL
LIN {X 0,Y 274.878,Z 435.612,A -85,B 0,C 180,E1 -18482.527,E2 -18482.527} C_VEL
LIN {X 0,Y 269.054,Z 423.117,A -85,B 0,C 180,E1 -18483.923,E2 -18483.923} C_VEL
LIN {X 0,Y 265.157,Z 415.615,A -85,B 0,C 180,E1 -18484.879,E2 -18484.879} C_VEL
LIN {X 0,Y 262.638,Z 410.948,A -85,B 0,C 180,E1 -18485.513,E2 -18485.513} C_VEL
LIN {X 0,Y 260.88,Z 407.286,A -85,B 0,C 180,E1 -18486.004,E2 -18486.004} C_VEL
LIN {X 0,Y 259.006,Z 399.549,A -85,B 0,C 180,E1 -18489.48,E2 -18489.48} C_VEL
LIN {X 0,Y 256.569,Z 391.376,A -85,B 0,C 180,E1 -18493.551,E2 -18493.551} C_VEL
LIN {X 0,Y 256.069,Z 389.588,A -85,B 0,C 180,E1 -18494.566,E2 -18494.566} C_VEL
LIN {X 0,Y 256.127,Z 389.582,A -85,B 0,C 180,E1 -18498.811,E2 -18498.811} C_VEL
LIN {X 0,Y 256.152,Z 389.571,A -85,B 0,C 180,E1 -18502.871,E2 -18502.871} C_VEL
LIN {X 0,Y 256.081,Z 389.577,A -85,B 0,C 180,E1 -18506.709,E2 -18506.709} C_VEL
LIN {X 0,Y 256.137,Z 389.576,A -85,B 0,C 180,E1 -18511.403,E2 -18511.403} C_VEL
LIN {X 0,Y 256.162,Z 389.575,A -85,B 0,C 180,E1 -18515.699,E2 -18515.699} C_VEL
LIN {X 0,Y 256.161,Z 389.567,A -85,B 0,C 180,E1 -18519.105,E2 -18519.105} C_VEL
LIN {X 0,Y 256.274,Z 389.556,A -85,B 0,C 180,E1 -18524.084,E2 -18524.084} C_VEL
LIN {X 0,Y 256.304,Z 389.553,A -85,B 0,C 180,E1 -18528.934,E2 -18528.934} C_VEL
LIN {X 0,Y 256.532,Z 389.516,A -85,B 0,C 180,E1 -18532.127,E2 -18532.127} C_VEL
LIN {X 0,Y 256.709,Z 389.498,A -85,B 0,C 180,E1 -18538.432,E2 -18538.432} C_VEL
LIN {X 0,Y 256.71,Z 389.498,A -85,B 0,C 180,E1 -18541.569,E2 -18541.569} C_VEL
LIN {X 0,Y 256.466,Z 389.528,A -85,B 0,C 180,E1 -18546.728,E2 -18546.728} C_VEL
LIN {X 0,Y 256.422,Z 389.545,A -85,B 0,C 180,E1 -18549.466,E2 -18549.466} C_VEL
LIN {X 0,Y 256.247,Z 389.566,A -85,B 0,C 180,E1 -18554.291,E2 -18554.291} C_VEL
LIN {X 0,Y 256.213,Z 389.566,A -85,B 0,C 180,E1 -18557.562,E2 -18557.562} C_VEL
LIN {X 0,Y 256.195,Z 389.566,A -85,B 0,C 180,E1 -18561.144,E2 -18561.144} C_VEL
LIN {X 0,Y 256.185,Z 389.571,A -85,B 0,C 180,E1 -18565.139,E2 -18565.139} C_VEL
LIN {X 0,Y 256.11,Z 389.581,A -85,B 0,C 180,E1 -18569.601,E2 -18569.601} C_VEL
LIN {X 0,Y 256.083,Z 389.57,A -85,B 0,C 180,E1 -18573.291,E2 -18573.291} C_VEL
LIN {X 0,Y 256.161,Z 389.694,A -85,B 0,C 180,E1 -18577.005,E2 -18577.005} C_VEL
LIN {X 0,Y 256.336,Z 390.534,A -85,B 0,C 180,E1 -18577.162,E2 -18577.162} C_VEL
LIN {X 0,Y 257.662,Z 393.167,A -85,B 0,C 180,E1 -18577.538,E2 -18577.538} C_VEL
LIN {X 0,Y 259.181,Z 394.898,A -85,B 0,C 180,E1 -18577.912,E2 -18577.912} C_VEL
LIN {X 0,Y 261.375,Z 398.305,A -85,B 0,C 180,E1 -18578.474,E2 -18578.474} C_VEL
LIN {X 0,Y 267.672,Z 408.719,A -85,B 0,C 180,E1 -18580.022,E2 -18580.022} C_VEL
LIN {X 0,Y 274.355,Z 421.316,A -85,B 0,C 180,E1 -18581.602,E2 -18581.602} C_VEL
LIN {X 0,Y 280.669,Z 434.706,A -85,B 0,C 180,E1 -18583.036,E2 -18583.036} C_VEL
LIN {X 0,Y 278.057,Z 495.359,A -85,B 0,C 180,E1 -18584.612,E2 -18584.612} C_VEL
LIN {X 0,Y 276.914,Z 508.969,A -85,B 0,C 180,E1 -18585.255,E2 -18585.255} C_VEL
LIN {X 0,Y 275.43,Z 520.947,A -85,B 0,C 180,E1 -18586.093,E2 -18586.093} C_VEL
LIN {X 0,Y 273.356,Z 533.571,A -85,B 0,C 180,E1 -18587.306,E2 -18587.306} C_VEL
LIN {X 0,Y 270.963,Z 545.227,A -85,B 0,C 180,E1 -18588.78,E2 -18588.78} C_VEL
LIN {X 0,Y 268.604,Z 555.149,A -85,B 0,C 180,E1 -18590.375,E2 -18590.375} C_VEL
LIN {X 0,Y 266.128,Z 564.116,A -85,B 0,C 180,E1 -18592.171,E2 -18592.171} C_VEL
LIN {X 0,Y 263.338,Z 573.37,A -85,B 0,C 180,E1 -18594.518,E2 -18594.518} C_VEL
LIN {X 0,Y 260.956,Z 580.764,A -85,B 0,C 180,E1 -18596.917,E2 -18596.917} C_VEL
LIN {X 0,Y 259.195,Z 585.827,A -85,B 0,C 180,E1 -18598.991,E2 -18598.991} C_VEL
LIN {X 0,Y 257.487,Z 590.569,A -85,B 0,C 180,E1 -18601.481,E2 -18601.481} C_VEL
LIN {X 0,Y 256.175,Z 594.055,A -85,B 0,C 180,E1 -18603.964,E2 -18603.964} C_VEL
LIN {X 0,Y 255.476,Z 595.76,A -85,B 0,C 180,E1 -18605.63,E2 -18605.63} C_VEL
LIN {X 0,Y 254.899,Z 597.03,A -85,B 0,C 180,E1 -18607.294,E2 -18607.294} C_VEL
LIN {X 0,Y 254.316,Z 598.131,A -85,B 0,C 180,E1 -18609.984,E2 -18609.984} C_VEL
LIN {X 0,Y 253.979,Z 598.159,A -85,B 0,C 180,E1 -18612.279,E2 -18612.279} C_VEL
LIN {X 0,Y 253.892,Z 597.703,A -85,B 0,C 180,E1 -18613.93,E2 -18613.93} C_VEL
LIN {X 0,Y 253.952,Z 596.759,A -85,B 0,C 180,E1 -18615.608,E2 -18615.608} C_VEL
LIN {X 0,Y 254.031,Z 595.451,A -85,B 0,C 180,E1 -18617.213,E2 -18617.213} C_VEL
LIN {X 0,Y 254.363,Z 592.638,A -85,B 0,C 180,E1 -18619.654,E2 -18619.654} C_VEL
LIN {X 0,Y 254.894,Z 588.779,A -85,B 0,C 180,E1 -18622.076,E2 -18622.076} C_VEL
LIN {X 0,Y 255.569,Z 583.786,A -85,B 0,C 180,E1 -18624.477,E2 -18624.477} C_VEL
LIN {X 0,Y 256.527,Z 577.503,A -85,B 0,C 180,E1 -18626.859,E2 -18626.859} C_VEL
LIN {X 0,Y 257.783,Z 569.647,A -85,B 0,C 180,E1 -18629.219,E2 -18629.219} C_VEL
LIN {X 0,Y 259.076,Z 561.613,A -85,B 0,C 180,E1 -18631.166,E2 -18631.166} C_VEL
LIN {X 0,Y 260.624,Z 551.802,A -85,B 0,C 180,E1 -18633.092,E2 -18633.092} C_VEL
LIN {X 0,Y 262.12,Z 540.9,A -85,B 0,C 180,E1 -18634.806,E2 -18634.806} C_VEL
LIN {X 0,Y 263.483,Z 530.19,A -85,B 0,C 180,E1 -18636.125,E2 -18636.125} C_VEL
LIN {X 0,Y 264.803,Z 517.325,A -85,B 0,C 180,E1 -18637.338,E2 -18637.338} C_VEL
LIN {X 0,Y 265.708,Z 505.156,A -85,B 0,C 180,E1 -18638.173,E2 -18638.173} C_VEL
LIN {X 0,Y 266.27,Z 492.948,A -85,B 0,C 180,E1 -18638.729,E2 -18638.729} C_VEL
LIN {X 0,Y 268.321,Z 421.577,A -85,B 0,C 180,E1 -18640.633,E2 -18640.633} C_VEL
LIN {X 0,Y 262.818,Z 405.261,A -85,B 0,C 180,E1 -18641.594,E2 -18641.594} C_VEL
LIN {X 0,Y 258.351,Z 394.719,A -85,B 0,C 180,E1 -18642.325,E2 -18642.325} C_VEL
LIN {X 0,Y 256.46,Z 390.506,A -85,B 0,C 180,E1 -18642.636,E2 -18642.636} C_VEL
LIN {X 0,Y 256.28,Z 389.566,A -85,B 0,C 180,E1 -18642.723,E2 -18642.723} C_VEL
LIN {X 0,Y 256.287,Z 389.562,A -85,B 0,C 180,E1 -18646.302,E2 -18646.302} C_VEL
LIN {X 0,Y 256.161,Z 389.578,A -85,B 0,C 180,E1 -18651.119,E2 -18651.119} C_VEL
LIN {X 0,Y 256.191,Z 389.567,A -85,B 0,C 180,E1 -18655.138,E2 -18655.138} C_VEL
LIN {X 0,Y 256.116,Z 389.583,A -85,B 0,C 180,E1 -18659.599,E2 -18659.599} C_VEL
LIN {X 0,Y 256.069,Z 389.589,A -85,B 0,C 180,E1 -18663.292,E2 -18663.292} C_VEL
LIN {X 0,Y 256.116,Z 389.581,A -85,B 0,C 180,E1 -18667.27,E2 -18667.27} C_VEL
LIN {X 0,Y 256.055,Z 389.586,A -85,B 0,C 180,E1 -18671.202,E2 -18671.202} C_VEL
LIN {X 0,Y 256.061,Z 389.585,A -85,B 0,C 180,E1 -18675.528,E2 -18675.528} C_VEL
LIN {X 0,Y 256.054,Z 389.588,A -85,B 0,C 180,E1 -18678.796,E2 -18678.796} C_VEL
LIN {X 0,Y 256.128,Z 389.577,A -85,B 0,C 180,E1 -18682.866,E2 -18682.866} C_VEL
LIN {X 0,Y 256.065,Z 389.589,A -85,B 0,C 180,E1 -18686.706,E2 -18686.706} C_VEL
LIN {X 0,Y 256.11,Z 389.578,A -85,B 0,C 180,E1 -18690.399,E2 -18690.399} C_VEL
LIN {X 0,Y 256.184,Z 389.571,A -85,B 0,C 180,E1 -18694.861,E2 -18694.861} C_VEL
LIN {X 0,Y 256.163,Z 389.575,A -85,B 0,C 180,E1 -18699.104,E2 -18699.104} C_VEL
LIN {X 0,Y 256.295,Z 389.552,A -85,B 0,C 180,E1 -18704.084,E2 -18704.084} C_VEL
LIN {X 0,Y 256.292,Z 389.556,A -85,B 0,C 180,E1 -18708.933,E2 -18708.933} C_VEL
LIN {X 0,Y 256.51,Z 389.528,A -85,B 0,C 180,E1 -18712.126,E2 -18712.126} C_VEL
LIN {X 0,Y 256.494,Z 389.53,A -85,B 0,C 180,E1 -18716.858,E2 -18716.858} C_VEL
LIN {X 0,Y 256.759,Z 389.487,A -85,B 0,C 180,E1 -18720,E2 -18720} C_VEL
LIN {X 0,Y 256.503,Z 389.519,A -85,B 0,C 180,E1 -18723.019,E2 -18723.019} C_VEL
LIN {X 0,Y 255.776,Z 389.624,A -85,B 0,C 180,E1 -18724.329,E2 -18724.329} C_VEL
LIN {X 0,Y 252.935,Z 389.989,A -85,B 0,C 180,E1 -18726.466,E2 -18726.466} C_VEL
LIN {X 0,Y 249.686,Z 390.385,A -85,B 0,C 180,E1 -18729.096,E2 -18729.096} C_VEL
LIN {X 0,Y 249.308,Z 390.425,A -85,B 0,C 180,E1 -18730.006,E2 -18730.006} C_VEL
LIN {X 0,Y 249.196,Z 390.444,A -85,B 0,C 180,E1 -18734.704,E2 -18734.704} C_VEL
LIN {X 0,Y 249.134,Z 390.448,A -85,B 0,C 180,E1 -18738.077,E2 -18738.077} C_VEL
LIN {X 0,Y 249.082,Z 390.457,A -85,B 0,C 180,E1 -18741.518,E2 -18741.518} C_VEL
LIN {X 0,Y 249.126,Z 390.451,A -85,B 0,C 180,E1 -18745.482,E2 -18745.482} C_VEL
LIN {X 0,Y 249.082,Z 390.457,A -85,B 0,C 180,E1 -18748.995,E2 -18748.995} C_VEL
LIN {X 0,Y 249.032,Z 390.466,A -85,B 0,C 180,E1 -18752.425,E2 -18752.425} C_VEL
LIN {X 0,Y 249.072,Z 390.463,A -85,B 0,C 180,E1 -18756.338,E2 -18756.338} C_VEL
LIN {X 0,Y 249.074,Z 390.463,A -85,B 0,C 180,E1 -18760.464,E2 -18760.464} C_VEL
LIN {X 0,Y 249.019,Z 390.467,A -85,B 0,C 180,E1 -18764.875,E2 -18764.875} C_VEL
LIN {X 0,Y 249.049,Z 390.463,A -85,B 0,C 180,E1 -18767.371,E2 -18767.371} C_VEL
LIN {X 0,Y 249.05,Z 390.465,A -85,B 0,C 180,E1 -18771.625,E2 -18771.625} C_VEL
LIN {X 0,Y 249.117,Z 390.463,A -85,B 0,C 180,E1 -18774.165,E2 -18774.165} C_VEL
LIN {X 0,Y 251.187,Z 400.41,A -85,B 0,C 180,E1 -18777.887,E2 -18777.887} C_VEL
LIN {X 0,Y 252.911,Z 408.831,A -85,B 0,C 180,E1 -18780.911,E2 -18780.911} C_VEL
LIN {X 0,Y 255.727,Z 417.665,A -85,B 0,C 180,E1 -18781.461,E2 -18781.461} C_VEL
LIN {X 0,Y 260.922,Z 460.759,A -85,B 0,C 180,E1 -18783.215,E2 -18783.215} C_VEL
LIN {X 0,Y 259.183,Z 517.369,A -85,B 0,C 180,E1 -18784.772,E2 -18784.772} C_VEL
LIN {X 0,Y 258.351,Z 530.729,A -85,B 0,C 180,E1 -18785.437,E2 -18785.437} C_VEL
LIN {X 0,Y 257.136,Z 542.947,A -85,B 0,C 180,E1 -18786.333,E2 -18786.333} C_VEL
LIN {X 0,Y 255.593,Z 555.274,A -85,B 0,C 180,E1 -18787.573,E2 -18787.573} C_VEL
LIN {X 0,Y 253.992,Z 565.612,A -85,B 0,C 180,E1 -18788.918,E2 -18788.918} C_VEL
LIN {X 0,Y 252.384,Z 576.356,A -85,B 0,C 180,E1 -18790.691,E2 -18790.691} C_VEL
LIN {X 0,Y 250.871,Z 585.847,A -85,B 0,C 180,E1 -18792.643,E2 -18792.643} C_VEL
LIN {X 0,Y 249.528,Z 594.615,A -85,B 0,C 180,E1 -18794.899,E2 -18794.899} C_VEL
LIN {X 0,Y 248.311,Z 602.177,A -85,B 0,C 180,E1 -18797.329,E2 -18797.329} C_VEL
LIN {X 0,Y 247.524,Z 609.156,A -85,B 0,C 180,E1 -18800.192,E2 -18800.192} C_VEL
LIN {X 0,Y 247.175,Z 613.735,A -85,B 0,C 180,E1 -18802.649,E2 -18802.649} C_VEL
LIN {X 0,Y 247.01,Z 617.191,A -85,B 0,C 180,E1 -18805.104,E2 -18805.104} C_VEL
LIN {X 0,Y 247.066,Z 618.904,A -85,B 0,C 180,E1 -18806.739,E2 -18806.739} C_VEL
LIN {X 0,Y 247.082,Z 620.196,A -85,B 0,C 180,E1 -18808.37,E2 -18808.37} C_VEL
LIN {X 0,Y 247.096,Z 621.082,A -85,B 0,C 180,E1 -18810,E2 -18810} C_VEL
LIN {X 0,Y 247.049,Z 621.547,A -85,B 0,C 180,E1 -18811.63,E2 -18811.63} C_VEL
LIN {X 0,Y 246.995,Z 621.582,A -85,B 0,C 180,E1 -18813.262,E2 -18813.262} C_VEL
LIN {X 0,Y 246.989,Z 621.14,A -85,B 0,C 180,E1 -18815.182,E2 -18815.182} C_VEL
LIN {X 0,Y 247.203,Z 619.375,A -85,B 0,C 180,E1 -18818.172,E2 -18818.172} C_VEL
LIN {X 0,Y 247.595,Z 617.811,A -85,B 0,C 180,E1 -18819.806,E2 -18819.806} C_VEL
LIN {X 0,Y 248.404,Z 614.699,A -85,B 0,C 180,E1 -18822.251,E2 -18822.251} C_VEL
LIN {X 0,Y 249.745,Z 610.563,A -85,B 0,C 180,E1 -18824.671,E2 -18824.671} C_VEL
LIN {X 0,Y 251.833,Z 604.278,A -85,B 0,C 180,E1 -18827.457,E2 -18827.457} C_VEL
LIN {X 0,Y 254.092,Z 597.26,A -85,B 0,C 180,E1 -18829.879,E2 -18829.879} C_VEL
LIN {X 0,Y 256.629,Z 589.067,A -85,B 0,C 180,E1 -18832.12,E2 -18832.12} C_VEL
LIN {X 0,Y 259.302,Z 580.436,A -85,B 0,C 180,E1 -18833.988,E2 -18833.988} C_VEL
LIN {X 0,Y 262.256,Z 569.849,A -85,B 0,C 180,E1 -18835.815,E2 -18835.815} C_VEL
LIN {X 0,Y 264.858,Z 559.365,A -85,B 0,C 180,E1 -18837.24,E2 -18837.24} C_VEL
LIN {X 0,Y 267.346,Z 547.777,A -85,B 0,C 180,E1 -18838.454,E2 -18838.454} C_VEL
LIN {X 0,Y 269.356,Z 535.804,A -85,B 0,C 180,E1 -18839.396,E2 -18839.396} C_VEL
LIN {X 0,Y 270.965,Z 522.653,A -85,B 0,C 180,E1 -18840.127,E2 -18840.127} C_VEL
LIN {X 0,Y 271.936,Z 509.603,A -85,B 0,C 180,E1 -18840.569,E2 -18840.569} C_VEL
LIN {X 0,Y 273.726,Z 464.12,A -85,B 0,C 180,E1 -18841.775,E2 -18841.775} C_VEL
LIN {X 0,Y 271.168,Z 446.806,A -85,B 0,C 180,E1 -18842.76,E2 -18842.76} C_VEL
LIN {X 0,Y 269.536,Z 438.559,A -85,B 0,C 180,E1 -18843.312,E2 -18843.312} C_VEL
LIN {X 0,Y 262.732,Z 424.09,A -85,B 0,C 180,E1 -18845.023,E2 -18845.023} C_VEL
LIN {X 0,Y 255.895,Z 411.25,A -85,B 0,C 180,E1 -18846.826,E2 -18846.826} C_VEL
LIN {X 0,Y 253.596,Z 406.869,A -85,B 0,C 180,E1 -18847.485,E2 -18847.485} C_VEL
LIN {X 0,Y 251.679,Z 399.356,A -85,B 0,C 180,E1 -18851.065,E2 -18851.065} C_VEL
LIN {X 0,Y 249.558,Z 392.414,A -85,B 0,C 180,E1 -18854.751,E2 -18854.751} C_VEL
LIN {X 0,Y 249.03,Z 390.463,A -85,B 0,C 180,E1 -18855.956,E2 -18855.956} C_VEL
LIN {X 0,Y 249.081,Z 390.455,A -85,B 0,C 180,E1 -18859.624,E2 -18859.624} C_VEL
LIN {X 0,Y 249.072,Z 390.453,A -85,B 0,C 180,E1 -18863.662,E2 -18863.662} C_VEL
LIN {X 0,Y 249.036,Z 390.462,A -85,B 0,C 180,E1 -18867.844,E2 -18867.844} C_VEL
LIN {X 0,Y 249.096,Z 390.452,A -85,B 0,C 180,E1 -18871.338,E2 -18871.338} C_VEL
LIN {X 0,Y 249.147,Z 390.443,A -85,B 0,C 180,E1 -18874.968,E2 -18874.968} C_VEL
LIN {X 0,Y 249.106,Z 390.456,A -85,B 0,C 180,E1 -18880.211,E2 -18880.211} C_VEL
LIN {X 0,Y 249.218,Z 390.431,A -85,B 0,C 180,E1 -18883.621,E2 -18883.621} C_VEL
LIN {X 0,Y 249.247,Z 390.429,A -85,B 0,C 180,E1 -18888.617,E2 -18888.617} C_VEL
LIN {X 0,Y 249.474,Z 390.396,A -85,B 0,C 180,E1 -18891.903,E2 -18891.903} C_VEL
LIN {X 0,Y 249.431,Z 390.404,A -85,B 0,C 180,E1 -18896.77,E2 -18896.77} C_VEL
LIN {X 0,Y 249.73,Z 390.378,A -85,B 0,C 180,E1 -18900,E2 -18900} C_VEL
LIN {X 0,Y 249.431,Z 390.402,A -85,B 0,C 180,E1 -18903.231,E2 -18903.231} C_VEL
LIN {X 0,Y 249.436,Z 390.403,A -85,B 0,C 180,E1 -18906.712,E2 -18906.712} C_VEL
LIN {X 0,Y 249.339,Z 390.427,A -85,B 0,C 180,E1 -18909.737,E2 -18909.737} C_VEL
LIN {X 0,Y 249.197,Z 390.444,A -85,B 0,C 180,E1 -18914.704,E2 -18914.704} C_VEL
LIN {X 0,Y 249.144,Z 390.451,A -85,B 0,C 180,E1 -18918.077,E2 -18918.077} C_VEL
LIN {X 0,Y 249.133,Z 390.448,A -85,B 0,C 180,E1 -18921.515,E2 -18921.515} C_VEL
LIN {X 0,Y 249.127,Z 390.454,A -85,B 0,C 180,E1 -18925.483,E2 -18925.483} C_VEL
LIN {X 0,Y 249.08,Z 390.461,A -85,B 0,C 180,E1 -18928.994,E2 -18928.994} C_VEL
LIN {X 0,Y 249.034,Z 390.46,A -85,B 0,C 180,E1 -18932.426,E2 -18932.426} C_VEL
LIN {X 0,Y 249.078,Z 390.446,A -85,B 0,C 180,E1 -18935.572,E2 -18935.572} C_VEL
LIN {X 0,Y 250.015,Z 393.147,A -85,B 0,C 180,E1 -18935.894,E2 -18935.894} C_VEL
LIN {X 0,Y 252.234,Z 395.837,A -85,B 0,C 180,E1 -18936.492,E2 -18936.492} C_VEL
LIN {X 0,Y 254.47,Z 399.265,A -85,B 0,C 180,E1 -18937.106,E2 -18937.106} C_VEL
LIN {X 0,Y 260.066,Z 407.801,A -85,B 0,C 180,E1 -18938.566,E2 -18938.566} C_VEL
LIN {X 0,Y 267.468,Z 421.233,A -85,B 0,C 180,E1 -18940.421,E2 -18940.421} C_VEL
LIN {X 0,Y 274.885,Z 436.796,A -85,B 0,C 180,E1 -18942.202,E2 -18942.202} C_VEL
LIN {X 0,Y 272.283,Z 495.646,A -85,B 0,C 180,E1 -18943.763,E2 -18943.763} C_VEL
LIN {X 0,Y 271.062,Z 509.428,A -85,B 0,C 180,E1 -18944.423,E2 -18944.423} C_VEL
LIN {X 0,Y 269.556,Z 521.145,A -85,B 0,C 180,E1 -18945.256,E2 -18945.256} C_VEL
LIN {X 0,Y 267.512,Z 533.08,A -85,B 0,C 180,E1 -18946.4,E2 -18946.4} C_VEL
LIN {X 0,Y 265.14,Z 544.475,A -85,B 0,C 180,E1 -18947.845,E2 -18947.845} C_VEL
LIN {X 0,Y 262.529,Z 554.93,A -85,B 0,C 180,E1 -18949.521,E2 -18949.521} C_VEL
LIN {X 0,Y 259.741,Z 564.716,A -85,B 0,C 180,E1 -18951.515,E2 -18951.515} C_VEL
LIN {X 0,Y 257.224,Z 572.646,A -85,B 0,C 180,E1 -18953.541,E2 -18953.541} C_VEL
LIN {X 0,Y 254.751,Z 579.887,A -85,B 0,C 180,E1 -18955.857,E2 -18955.857} C_VEL
LIN {X 0,Y 252.772,Z 585.459,A -85,B 0,C 180,E1 -18958.112,E2 -18958.112} C_VEL
LIN {X 0,Y 250.774,Z 590.652,A -85,B 0,C 180,E1 -18960.819,E2 -18960.819} C_VEL
LIN {X 0,Y 249.439,Z 594.015,A -85,B 0,C 180,E1 -18963.205,E2 -18963.205} C_VEL
LIN {X 0,Y 248.679,Z 595.816,A -85,B 0,C 180,E1 -18964.918,E2 -18964.918} C_VEL
LIN {X 0,Y 248.005,Z 597.151,A -85,B 0,C 180,E1 -18966.626,E2 -18966.626} C_VEL
LIN {X 0,Y 247.274,Z 598.466,A -85,B 0,C 180,E1 -18969.708,E2 -18969.708} C_VEL
LIN {X 0,Y 246.951,Z 598.534,A -85,B 0,C 180,E1 -18971.757,E2 -18971.757} C_VEL
LIN {X 0,Y 246.812,Z 598.146,A -85,B 0,C 180,E1 -18973.456,E2 -18973.456} C_VEL
LIN {X 0,Y 246.847,Z 597.12,A -85,B 0,C 180,E1 -18975.473,E2 -18975.473} C_VEL
LIN {X 0,Y 247.059,Z 594.398,A -85,B 0,C 180,E1 -18978.514,E2 -18978.514} C_VEL
LIN {X 0,Y 247.553,Z 591.025,A -85,B 0,C 180,E1 -18981.017,E2 -18981.017} C_VEL
